    2:
        IF fbMotionDriveStateMachine.WatchDogTimeOut THEN
            nTestStep := nTestStep + 1;
        END_IF
    3:
        AssertEquals_INT(	Expected:=expectedMoveState,
                            Actual:=fbMotionDriveStateMachine.State,
                            Message:='Drive Machine state must be ERROR #1');
        AssertTrue(Condition := fbMotionDriveStateMachine.Error, Message := 'Motion Drive state machine must be in error state #2');
        nTestStep := nTestStep + 1;
        TEST_FINISHED();
END_CASE

fbMotionDriveStateMachine();
fbTestTimer();

IF fbTestTimer.Q THEN
    AssertTrue(Condition := FALSE, Message := CONCAT('Timed out at step: ', TO_STRING(nTestStep)));
    TEST_FINISHED();
END_IF
END_METHOD

METHOD PRIVATE GIvenStartedStatedAndErrorThenGotoErrorState_Test6
VAR_INST
    fbMotionDriveStateMachine : FB_MotionDriveStateMachine(
		stMotionCommand := THIS^.stMotionCommand[6],
		iMotionAxis:=THIS^.fbMotionAxisNC[6], 
		iMoveRequest:=THIS^.fbMoveRequest[6],
		iMotionLogger := THIS^.fbMotionLogger[6]
	);
    expectedMoveState : E_MoveState := E_MoveState.ERROR;

    nTestStep : INT;
END_VAR
TEST(__POUNAME());
CASE nTestStep OF
    0:
        fbMotionDriveStateMachine.State := E_MoveState.STARTED;
        fbMotionDriveStateMachine.StateMachine(Error:=TRUE);
        nTestStep := nTestStep + 1;
    1:
        AssertEquals_INT(	Expected:=expectedMoveState,
                            Actual:=fbMotionDriveStateMachine.State,
                            Message:='Drive Machine must be ERROR state #1');
        TEST_FINISHED();
END_CASE

fbMotionDriveStateMachine();
END_METHOD

END_FUNCTION_BLOCK

// ---- Test/TestDouble/FB_MotionAxisNC_TestDouble.TcPOU
FUNCTION_BLOCK FB_MotionAxisNC_TestDouble IMPLEMENTS I_MotionAxis
VAR

    iHome : I_Home;
    iHalt : I_Halt;
    iPower : I_Power;
    iReset : I_Reset;
    iMoveAbsolute : I_MoveAbsolute;
    iReadParameter : I_ReadParameter;
    iWriteParameter  : I_WriteParameter;
    iParamSaveRestore: I_ParamsSaveRestore;
    iEncoderScaling : I_EncoderScaling;
    iAxisStatus : I_AxisStatus;
    iBacklashCompensation : I_BacklashCompensation;

    bError: BOOL;
    nErrorID: UDINT;
    sMessage : T_MAXSTRING;
    stMotionAxisStatus : ST_AxisStatus;
END_VAR

METHOD AxisEnabled : BOOL
END_METHOD

(*
    Handle positive/negative backlash compensation
    User needs to set the direction of backlash from the sign of the compensation value
    Backlash compensation is disabled during referencing (homing).
    When direction is positive/negative, further movement in the negative/positive direction not compensated
    further movement in the negative/positive direction will be compensated
*)
METHOD BacklashCompensation
VAR_INPUT
    Enable	: BOOL := FALSE;
    RampVelo	: LREAL;
END_VAR
END_METHOD

METHOD ClearHaltStatus
END_METHOD

{warning 'Add method implementation '}
METHOD ClearHomeStatus
END_METHOD

{warning 'Add method implementation '}
METHOD ClearMoveAbsoluteStatus
END_METHOD

METHOD ClearResetStatus
END_METHOD

METHOD DisablePower
END_METHOD

METHOD DriveCommands
VAR_INPUT
    HomeCmd	: BOOL;
    NewMoveReq	: BOOL;
    EnableMode	: E_StageEnableMode;
END_VAR
END_METHOD

METHOD Halt
VAR_INPUT
    Deceleration	: LREAL := 0;
    Jerk	: LREAL := 0;
    BufferMode	: MC_BufferMode := MC_BufferMode.MC_Aborting;
END_VAR
END_METHOD

METHOD Home
VAR_INPUT
    Position        : LREAL         := DEFAULT_HOME_POSITION;
    BufferMode      : MC_BufferMode;
 	HomeMode: INT :=E_EpicsHomeCmd.NONE;
END_VAR
END_METHOD

{warning 'Add method implementation '}
METHOD HomeAbortRecovery
END_METHOD

METHOD MoveAbsolute
VAR_INPUT
    Position	: LREAL;
    Velocity	: LREAL;
    Acceleration	: LREAL := 0;
    Deceleration	: LREAL := 0;
    Jerk	: LREAL := 0;
    BufferMode	: MC_BufferMode := MC_BufferMode.MC_Aborting;
END_VAR
END_METHOD

METHOD Power
VAR_INPUT
    Enable	: BOOL;
    Enable_Positive	: BOOL;
    Enable_Negative	: BOOL;
    Override	: LREAL;
    BufferMode	: MC_BufferMode;
END_VAR
END_METHOD

METHOD ReadAxisParams
VAR_INPUT
    Enable	: BOOL;
    RefreshDelay	: TIME;
END_VAR
END_METHOD

METHOD Reset
END_METHOD

METHOD SaveAxisParams
VAR_INPUT
    Enable	: BOOL;
END_VAR
END_METHOD

PROPERTY Status : REFERENCE TO ST_AxisStatus
GET
Status REF= stMotionAxisStatus;
END_GET
END_PROPERTY

END_FUNCTION_BLOCK

// ---- Test/TestDouble/FB_MotionAxisDS402_TestDouble.TcPOU
FUNCTION_BLOCK FB_MotionAxisDS402_TestDouble IMPLEMENTS I_MotionAxisDS402
VAR
    bError: BOOL;
    nErrorID: UDINT;
    sMessage : T_MAXSTRING;
    stMotionAxisStatus : ST_AxisStatus;
    bConfigDone : BOOL;
END_VAR

METHOD AxisEnabled : BOOL
END_METHOD

(*
    Handle positive/negative backlash compensation
    User needs to set the direction of backlash from the sign of the compensation value
    Backlash compensation is disabled during referencing (homing).
    When direction is positive/negative, further movement in the negative/positive direction not compensated
    further movement in the negative/positive direction will be compensated
*)
METHOD BacklashCompensation
VAR_INPUT
    Enable	: BOOL := FALSE;
    RampVelo	: LREAL;
END_VAR
END_METHOD

METHOD ClearHaltStatus
END_METHOD

{warning 'Add method implementation '}
METHOD ClearHomeStatus
END_METHOD

{warning 'Add method implementation '}
METHOD ClearMoveAbsoluteStatus
END_METHOD

METHOD ClearResetStatus
END_METHOD

PROPERTY ConfigDone : BOOL
GET
ConfigDone := bConfigDone;
END_GET
SET
bConfigDone := ConfigDone;
END_SET
END_PROPERTY

METHOD DisablePower
END_METHOD

METHOD DriveCommands
VAR_INPUT
    HomeCmd	: BOOL;
    NewMoveReq	: BOOL;
    EnableMode	: E_StageEnableMode;
END_VAR
END_METHOD

METHOD Halt
VAR_INPUT
    Deceleration	: LREAL := 0;
    Jerk	: LREAL := 0;
    BufferMode	: MC_BufferMode := MC_BufferMode.MC_Aborting;
END_VAR
END_METHOD

METHOD Home
VAR_INPUT
    Position        : LREAL         := DEFAULT_HOME_POSITION;
    BufferMode      : MC_BufferMode;
 	HomeMode: INT :=E_EpicsHomeCmd.NONE;
END_VAR
END_METHOD

METHOD ModeConfigDone : BOOL
VAR_INPUT
    Mode	: E_EpicsMotorCmd;
END_VAR
 ModeConfigDone :=  bConfigDone;
END_METHOD

METHOD ModeOfOperation : BOOL
VAR_INPUT
    RecentModeOfOperation	: E_DS402OpMode;
END_VAR
END_METHOD

METHOD MoveAbsolute
VAR_INPUT
    Position	: LREAL;
    Velocity	: LREAL;
    Acceleration	: LREAL := 0;
    Deceleration	: LREAL := 0;
    Jerk	: LREAL := 0;
    BufferMode	: MC_BufferMode := MC_BufferMode.MC_Aborting;
END_VAR
END_METHOD

METHOD Power
VAR_INPUT
    Enable	: BOOL;
    Enable_Positive	: BOOL;
    Enable_Negative	: BOOL;
    Override	: LREAL;
    BufferMode	: MC_BufferMode;
END_VAR
END_METHOD

METHOD ReadAxisParams
VAR_INPUT
    Enable	: BOOL;
    RefreshDelay	: TIME;
END_VAR
END_METHOD

METHOD Reset
END_METHOD

METHOD SaveAxisParams
VAR_INPUT
    Enable	: BOOL;
END_VAR
END_METHOD

PROPERTY Status : REFERENCE TO ST_AxisStatus
GET
Status REF= stMotionAxisStatus;
END_GET
END_PROPERTY

END_FUNCTION_BLOCK

// ---- Test/TestDouble/FB_MoveRequest_TestDouble.TcPOU
FUNCTION_BLOCK FB_MoveRequest_TestDouble IMPLEMENTS I_MoveRequest
VAR
    eEnableMode: E_StageEnableMode:=E_StageEnableMode.DURING_MOTION;
    bMoveCmd	: BOOL;
    bHomeCmd: BOOL;
    eHomeMode	: E_EpicsHomeCmd;
    bEnableDone : BOOL;
    bMoveOk: BOOL;
    bExecute : BOOL;
    stMotionRequestStatus : ST_MoveRequestStatus;
END_VAR

METHOD ClearMoveRequest
END_METHOD

METHOD ClearMoveRequestErrors
END_METHOD

PROPERTY EnableMode : ENUM_StageEnableMode
GET
END_GET
SET
END_SET
END_PROPERTY

PROPERTY INTERNAL EpicsMotorCommand : INT
GET
EpicsMotorCommand := stMotionRequestStatus.nCommand;
END_GET
SET
stMotionRequestStatus.nCommand := EpicsMotorCommand;
END_SET
END_PROPERTY

METHOD HaltMoveRequest : BOOL
VAR_INPUT
    Busy	: BOOL;
END_VAR
END_METHOD

METHOD InitMoveRequest
END_METHOD

METHOD IsValidHomeCmd : BOOL
VAR_INPUT
    CmdData : INT;
END_VAR
END_METHOD

METHOD MoveRequest
VAR_INPUT
    (* From Axis through the drive*)
    EnableDone	: BOOL;
    (* From Interlock through the drive*)
    MoveOk	: BOOL;
END_VAR
END_METHOD

METHOD MoveRequestCompleted
VAR_INPUT
    MoveDone	: BOOL;
    HomeDone	: BOOL;
END_VAR
END_METHOD

METHOD MoveRequestDone
VAR_INPUT
    Done	: BOOL;
END_VAR
END_METHOD

METHOD MoveRequestError
VAR_INPUT
    Error	: BOOL;
    ErrorId	: UDINT;
    ErrorMessage	: T_MAXSTRING;
END_VAR
END_METHOD

METHOD MoveResetDone
END_METHOD

METHOD ResetMoveEnable : BOOL
END_METHOD

METHOD ResetMoveRequest
END_METHOD

METHOD RestoreSettings
VAR_INPUT
    RestoreDone : BOOL;
    SavedPosition : LREAL;
END_VAR
END_METHOD

PROPERTY Status : REFERENCE TO ST_MoveRequestStatus
GET
Status REF= stMotionRequestStatus;
END_GET
END_PROPERTY

{warning 'Add method implementation '}
METHOD StopMoveRequest
END_METHOD

END_FUNCTION_BLOCK

// ---- Test/Orchetration/FB_MotionDrive_Test.TcPOU
FUNCTION_BLOCK FB_MotionDrive_Test EXTENDS FB_TestSuite
VAR
	stMotionCommand : ST_MotionCommand;
    stMotionStatus: ST_MotionStatus;
	stExMotionStatus : ST_ExtendedMotionStatus;
    fbAxis         : FB_MotionAxisNC_TestDouble;        
    fbInterlocks   : FB_MotionInterlocksLimSw_TestDouble;  
    fbLogger       : FB_MotionLogger_TestDouble;      
    fbMoveRequest  : FB_MoveRequest_TestDouble;        
    fbStateMachine : FB_StateMachine_TestDouble;      
    fbBrake        : FB_Brake_TestDouble;              
END_VAR

NoCrashTest();

METHOD PRIVATE NoCrashTest
VAR_INST
	fbMotionDrive : FB_MotionDrive(	
		stMotionCommand :=stMotionCommand,
		stMotionStatus:=stMotionStatus,
		stExMotionStatus :=stExMotionStatus,
		iInterlocks :=fbInterlocks,
		iLogger :=fbLogger,
		iAxis:=fbAxis,
		iMoveRequest :=fbMoveRequest,
		iStateMachine :=fbStateMachine,
		iBrake :=fbBrake
	);


END_VAR
(*This method is called cyclicly in the fbMotionDrive *)
TEST(__POUNAME());
fbMotionDrive();
TEST_FINISHED();
END_METHOD

END_FUNCTION_BLOCK

// ---- Test/TestDouble/FB_MotionInterlocksLimSw_TestDouble.TcPOU
FUNCTION_BLOCK FB_MotionInterlocksLimSw_TestDouble IMPLEMENTS I_MotionInterlocks
VAR
END_VAR

METHOD AxisStatus
VAR_INPUT
    HomeBusy	: BOOL;
    PositiveDirection	: BOOL;
    NegativeDirection	: BOOL;
END_VAR
END_METHOD

METHOD DriveCommands
VAR_INPUT
    MoveEnable: BOOL;
    NewMoveReq : BOOL;
END_VAR
END_METHOD

PROPERTY Error : BOOL
GET
END_GET
END_PROPERTY

PROPERTY ErrorID : UDINT
GET
END_GET
END_PROPERTY

PROPERTY InterlockEvent : BOOL
GET
END_GET
END_PROPERTY

PROPERTY LimHome : BOOL
GET
END_GET
END_PROPERTY

PROPERTY Message : T_MAXSTRING
GET
END_GET
END_PROPERTY

PROPERTY MoveBackwardEnabled : BOOL
GET
END_GET
END_PROPERTY

PROPERTY MoveForwardEnabled : BOOL
GET
END_GET
END_PROPERTY

PROPERTY MoveOk : BOOL
GET
END_GET
END_PROPERTY

PROPERTY PowerEnabled : BOOL
GET
END_GET
END_PROPERTY

METHOD Reset
END_METHOD

PROPERTY Warning : BOOL
GET
END_GET
END_PROPERTY

END_FUNCTION_BLOCK

// ---- Test/TestDouble/FB_StateMachine_TestDouble.TcPOU
FUNCTION_BLOCK FB_StateMachine_TestDouble IMPLEMENTS I_StateMachine
VAR
END_VAR

{warning 'Add property implementation'}
PROPERTY Idling : BOOL
GET
END_GET
END_PROPERTY

PROPERTY MoveState : E_MOVESTATE
GET
END_GET
END_PROPERTY

{warning 'Add method implementation '}
METHOD Reset
END_METHOD

METHOD StateMachine
VAR_INPUT
	Error : BOOL;
	InterlockEvent : BOOL;
END_VAR
END_METHOD

PROPERTY WatchDogStatus : BOOL
GET
END_GET
END_PROPERTY

PROPERTY WatchDogTimeOut : BOOL
GET
END_GET
END_PROPERTY

END_FUNCTION_BLOCK

// ---- POUs/FBs/Common/FB_MotionDrive.TcPOU
FUNCTION_BLOCK FB_MotionDrive IMPLEMENTS I_MotionDrive
VAR_INPUT
END_VAR
VAR_OUTPUT
END_VAR
VAR
   // EPICS Interface
    {attribute 'no_copy'}
    stMotionEpicsItf : REFERENCE TO ST_MotionEpicsItf;
    {attribute 'hide'}
    iMotionAxis: I_MotionAxis;
    {attribute 'hide'}
    iBrake 				: I_Brake;
    {attribute 'hide'}
    iMotionInterlocks	: I_MotionInterlocks;
    {attribute 'hide'}
    iMotionLogger 		: I_MotionLogger;
    {attribute 'hide'}
    eMoveMode : E_EpicsMotorCmd := E_EpicsMotorCmd.MOVE_ABSOLUTE;
    // Determines when we automatically enable the motor
    //{attribute 'hide'}
    eEnableMode: E_StageEnableMode:=E_StageEnableMode.DURING_MOTION;

    (* Shortcut Commands *)
    // Start a move to fPosition with fVelocity
    bMoveCmd: BOOL;
    // Start the homing routine
    {attribute 'pytmc' := '
        pv: PLC:bHomeCmd
        io: io
        field: DESC Start the homing routine
    '}
    bHomeCmd: BOOL;
    // Close or open loop operation ( DS402 Piezo axis )
    {attribute 'pytmc' := '
        pv: PLC:bServo
        io: io
        field: ZNAM FALSE
        field: ONAM TRUE
        field: DESC Used internally to reset errors
    '}
    bServo : BOOL;

    sName : STRING;
    {attribute 'hide'}
    eMoveState	: E_MoveState;
    {attribute 'hide'}
    bNewMoveReq : BOOL;
    {attribute 'hide'}
    bExecHome 	: BOOL;
    {attribute 'hide'}
    bExecMove 	: BOOL;
    {attribute 'hide'}
    rtMoveCmdShortcut	: R_TRIG;
    {attribute 'hide'}
    rtHomeCmdShortcut 	: R_TRIG;
    {attribute 'hide'}
    rtUserExec 			: R_TRIG;
    {attribute 'hide'}
    rtNewMoveReq 		: R_TRIG;
    {attribute 'hide'}
    rtTarget			: R_TRIG;
    {attribute 'hide'}
    rtHomed				: R_TRIG;
    {attribute 'hide'}
    rtValidExec 	: R_TRIG;
    {attribute 'hide'}
    rtReset 			: R_TRIG;
    {attribute 'hide'}
    ftStopExec 			: F_TRIG;
    {attribute 'hide'}
    ftError 			: F_TRIG;
    {attribute 'hide'}
    nCommandLocal: UINT;
    {attribute 'hide'}
    nCmdDataLocal: UINT;
    {attribute 'hide'}
    ftLocalStart : F_TRIG;
    {attribute 'hide'}
    bInitStart : BOOL;
    {attribute 'hide'}
    bLocalExec : BOOL;
    {attribute 'hide'}
    bEnableDone : BOOL;
    {attribute 'hide'}
    bPrepareDisable : BOOL;
    {attribute 'hide'}
    rtEnableMode : R_TRIG;
    {attribute 'hide'}
    rtStopExec : R_TRIG;
    {attribute 'hide'}
    rtInterlockEvent : R_TRIG;
    {attribute 'hide'}
    bCmdExecute : BOOL;
    {attribute 'hide'}
    bHaltAbort : BOOL;
    {attribute 'hide'}
    ftHaltAbort : F_TRIG;
    {attribute 'hide'}
    rtRestoreDone : R_TRIG;
    {attribute 'hide'}
    bHaltEvent : BOOL;
    // move state machine to error state in case a move command gets stuck after
    // the corresponding start signal was forwarded. the start signal should yeild a busy true response.
    // the move processing block may get stuck and return no errors. this is a contingency to make sure that reset would reinit all state machines.
    tonSyncTimer : TON;
    bLocalError : BOOL;
    bLocalMessage : T_MAXSTRING;
END_VAR

IF NOT __ISVALIDREF( THIS^.stMotionEpicsItf ) THEN
   RETURN;
END_IF
// Restore axis parameters
THIS^.RestoreSettings();

// catch high priority message
// an extended error message from FB_MotionLogger will display cyclic errors and warning
IF iMotionAxis.Error THEN
   stMotionEpicsItf.bError := iMotionAxis.Error;
   stMotionEpicsItf.nErrorId := iMotionAxis.ErrorID;
   stMotionEpicsItf.sErrorMessage := iMotionAxis.Message;
ELSIF iMotionInterlocks.Error THEN
   stMotionEpicsItf.bError := iMotionInterlocks.Error;
   stMotionEpicsItf.nErrorId := iMotionInterlocks.ErrorID;
   stMotionEpicsItf.sErrorMessage := iMotionInterlocks.Message;
ELSIF bLocalError THEN
   stMotionEpicsItf.bError := bLocalError;
   stMotionEpicsItf.sErrorMessage := bLocalMessage;
// Warnings have lowest priority
ELSIF iMotionInterlocks.Warning THEN
   stMotionEpicsItf.sErrorMessage := iMotionInterlocks.Message;
ELSE
       stMotionEpicsItf.bError := FALSE;
       stMotionEpicsItf.nErrorId := 0;
       stMotionEpicsItf.sErrorMessage := '';

END_IF

// Drive state machine
THIS^.StateMachine();
//
THIS^.PostHandling();
// update EPICS status
THIS^.UpdateParamAndStatus();

METHOD PUBLIC CallAfterInit
VAR_INPUT
    stMotionEpicsItf : REFERENCE TO ST_MotionEpicsItf;
    iBrake : I_Brake;
    iMotionInterlocks : I_MotionInterlocks;
    iMotionLogger : I_MotionLogger;
    iMotionAxis: I_MotionAxis;
END_VAR
THIS^.stMotionEpicsItf REF=stMotionEpicsItf;
THIS^.iMotionAxis := iMotionAxis;
THIS^.iMotionLogger:=iMotionLogger;
THIS^.iBrake:=iBrake;
THIS^.iMotionInterlocks:=iMotionInterlocks;
END_METHOD

METHOD ClearVars
VAR_INPUT
    Done : BOOL;
END_VAR
stMotionEpicsItf.bDone := Done;
stMotionEpicsItf.bBusy := FALSE;
// falling edge here when target is reached, move halted
stMotionEpicsItf.bExecute := FALSE;
THIS^.bLocalExec := FALSE;
// release the cmds
THIS^.bHomeCmd:=FALSE;
THIS^.bMoveCmd:=FALSE;
THIS^.binitStart := FALSE;
THIS^.bCmdExecute := FALSE;
THIS^.tonSyncTimer.IN:=FALSE;
END_METHOD

{warning 'Add property implementation'}
PROPERTY EnableMode : ENUM_StageEnableMode
GET
EnableMode := eEnableMode;
END_GET
SET
eEnableMode := EnableMode;
END_SET
END_PROPERTY

//FB_Init is always available implicitly and it is used primarily for initialization.
//The return value is not evaluated. For a specific influence, you can also declare the
//methods explicitly and provide additional code there with the standard initialization
//code. You can evaluate the return value.
METHOD FB_Init: BOOL
VAR_INPUT
    bInitRetains: BOOL; // TRUE: the retain variables are initialized (reset warm / reset cold)
    bInCopyCode: BOOL;  // TRUE: the instance will be copied to the copy code afterward (online change)
    stMotionEpicsItf : REFERENCE TO ST_MotionEpicsItf;
    iBrake : I_Brake;
    iMotionInterlocks : I_MotionInterlocks;
    iMotionLogger : I_MotionLogger;
    iMotionAxis: I_MotionAxis;
   // iLimSwStatus : I_LimSwStatus;
END_VAR
THIS^.stMotionEpicsItf REF=stMotionEpicsItf;
THIS^.iMotionAxis := iMotionAxis;
THIS^.iMotionLogger:=iMotionLogger;
THIS^.iBrake:=iBrake;
//THIS^.iLimSwStatus:=iLimSwStatus;
THIS^.iMotionInterlocks:=iMotionInterlocks;
END_METHOD

{attribute 'call_after_init'}
METHOD Instances
VAR_INPUT
END_VAR

VAR

END_VAR
// bMotionAxisNC  := __QUERYINTERFACE(iMotionAxisCommon, iMotionAxisNC) AND NOT __QUERYINTERFACE(iMotionAxisCommon,iMotionAxisCommonDS402);
// bMotionAxisNCDS402  := __QUERYINTERFACE(iMotionAxisCommon,iMotionAxisNCDS402) AND __QUERYINTERFACE(iMotionAxisCommon,iMotionAxisCommonDS402);
// bMotionAxisDS402  := __QUERYINTERFACE(iMotionAxisCommon, iMotionAxisDS402);
// bMotionInterlocks  := __QUERYINTERFACE(iMotionInterlocks,iMotionInterlocks) AND NOT __QUERYINTERFACE(iMotionInterlocks,iLimSw);
// bMotionInterlocksLimSw  := __QUERYINTERFACE(iMotionInterlocks,iMotionInterlocks) AND __QUERYINTERFACE(iMotionInterlocks,iLimSw);;
END_METHOD

{warning 'Add property implementation'}
PROPERTY Name : STRING
GET
Name := sName;
END_GET
SET
sName := Name;
END_SET
END_PROPERTY

{warning 'Add method implementation '}
METHOD PostHandling
// Move done, or aborted? prepare disable.
// we'll wait for axis to be in standstill and this state machine to be idling.
THIS^.bPrepareDisable S= (eEnableMode = E_StageEnableMode.DURING_MOTION ) AND THIS^.ftStopExec.Q;
//
// IF THIS^.stMotionEpicsItf.bReset THEN
//    // Relese motion cmds
//    THIS^.ClearVars(Done:=FALSE);
//  			THIS^.bLocalError := FALSE;
// 			THIS^.bLocalMessage := '';
//    // Forward general reset event
//    THIS^.iMotionAxis.Reset(Execute:= THIS^.stMotionEpicsItf.bReset);
//    THIS^.stMotionEpicsItf.bReset := FALSE;
// END_IF

// When reset is done axis is standstill
// safe to remove power
IF iMotionAxis.ResetDone THEN
    THIS^.stMotionEpicsItf.bEnable := FALSE;
END_IF

// Default is move absolute for state psotioner
IF THIS^.rtHomed.Q THEN
       stMotionEpicsItf.nCommand:=E_EpicsMotorCmd.MOVE_ABSOLUTE;
END_IF
// Halt is always a user stop but not an interlock event or a reset.
bHaltEvent S= ftStopExec.Q AND ((iMotionAxis.HomeBusy AND (nCommandLocal=10))
                            OR(iMotionAxis.MoveAbsoluteBusy AND (nCommandLocal=3)));
bHaltEvent R= THIS^.iMotionAxis.HaltDone OR THIS^.iMotionAxis.ResetDone;

THIS^.iMotionAxis.Halt(	Execute:=bHaltEvent,
                        Deceleration:=stMotionEpicsItf.fDeceleration);

//
THIS^.iMotionInterlocks.AxisStatus(
                            HomeBusy:=THIS^.iMotionAxis.HomeBusy,
                            PositiveDirection:=THIS^.iMotionAxis.PositiveMotionIsEnabled,
                            NegativeDirection:=THIS^.iMotionAxis.NegativeMotionIsEnabled );

// Forward drive commands to interlock blocks
THIS^.iMotionInterlocks.DriveCommands(Enable:=THIS^.stMotionEpicsItf.bEnable, NewMoveReq:=THIS^.bNewMoveReq, Reset:=THIS^.iMotionAxis.ResetDone);
// Forward Power block enable flags
THIS^.iMotionAxis.PowerEnables(Enable:=iMotionInterlocks.PowerEnabled,
                        Enable_Positive:=iMotionInterlocks.MoveForwardEnabled,
                        Enable_Negative:=iMotionInterlocks.MoveBackwardEnabled );

// Forward axis state to brake FB
THIS^.iBrake.AxisState := iMotionAxis.AxisState;

// Read Axis Parameter
THIS^.iMotionAxis.ReadAxisParams(Enable:=TRUE, RefreshDelay:=T#1S);

// Save and Restore
THIS^.iMotionAxis.SaveAxisParams(Enable:=TRUE);
END_METHOD

METHOD PreHandling
(*
  Check for the plc shortcut commands
  Used for testing or to circumvent motor record issues
  A request is process and qualified as a legitimate move after it clears interlocks checks
*)
rtMoveCmdShortcut(CLK:=THIS^.bMoveCmd);
rtHomeCmdShortcut(CLK:=THIS^.bHomeCmd);
// Execute on rising edge
IF rtMoveCmdShortcut.Q AND NOT stMotionEpicsItf.bExecute THEN
   stMotionEpicsItf.bExecute:=TRUE;
   stMotionEpicsItf.nCommand:=E_EpicsMotorCmd.MOVE_ABSOLUTE;
   // attempting to move an axis without homing first?
   IF iMotionAxis.HomeMode <> E_EpicsHomeCmd.NONE AND NOT iMotionAxis.HomeDone THEN
       stMotionEpicsItf.sErrorMessage:='Axis homing mode set, but homing routine pending';
   END_IF
ELSIF rtHomeCmdShortcut.Q AND NOT stMotionEpicsItf.bExecute THEN
       stMotionEpicsItf.nCommand:=E_EpicsMotorCmd.HOME;
       // Automatically fill the correct nCmdData for homing
       stMotionEpicsItf.nCmdData:=iMotionAxis.HomeMode;
       IF ( stMotionEpicsItf.nCmdData = E_EpicsHomeCmd.ABSOLUTE_SET )  OR ( stMotionEpicsItf.nCmdData = E_EpicsHomeCmd.NONE) THEN
       stMotionEpicsItf.bExecute:= FALSE;
       THIS^.bHomeCmd := FALSE;
    ELSE
        stMotionEpicsItf.bExecute:= TRUE;
    END_IF
END_IF

rtUserExec(CLK:=stMotionEpicsItf.bExecute);
bNewMoveReq S= rtUserExec.Q AND NOT iMotionAxis.Busy AND iMotionInterlocks.MoveOk;
// An axis or interlocks error will immediately invalidate this this request.
bNewMoveReq R= NOT stMotionEpicsItf.bExecute OR stMotionEpicsItf.bError;
bPrepareDisable R= bNewMoveReq;
//
rtNewMoveReq(CLK:=bNewMoveReq);
rtEnableMode(CLK:=(eEnableMode = E_StageEnableMode.DURING_MOTION));
// Handle auto-enable timing
CASE eEnableMode OF
   E_StageEnableMode.ALWAYS:
       stMotionEpicsItf.bEnable:=TRUE;
   E_StageEnableMode.DURING_MOTION:
       IF rtEnableMode.Q THEN
           stMotionEpicsItf.bEnable := FALSE;
       END_IF
       // Power interlock only enabled with a new move request
       IF rtNewMoveReq.Q THEN
           stMotionEpicsItf.bEnable S= bNewMoveReq (*iMotionInterlocks.SafetyReady*);
       END_IF
END_CASE
//
// Get a definitive bEnabled reading
THIS^.bEnableDone := THIS^.iMotionAxis.AxisEnabled(HomeCmd:=THIS^.bHomeCmd, NewMoveReq:=THIS^.bNewMoveReq);

// This is the output interlock check used to allow the requested move
bLocalExec:= stMotionEpicsItf.bExecute AND iMotionInterlocks.PowerEnabled AND THIS^.bEnableDone (*AND iMotionInterlocks.SafetyReady*);

bExecHome:=THIS^.bLocalExec AND stMotionEpicsItf.nCommand = 10;
bExecMove:=THIS^.bLocalExec AND NOT bExecHome;
//
// Transfer nCommand and nCmdData to local copies at rising edge of bExecute
// (avoid issues if nCommand or nCmdData are changed during a command)
rtValidExec(CLK:=(THIS^.bExecMove OR THIS^.bExecHome));
IF rtValidExec.Q THEN
 // used for jog, modulo, GearIn which are not implemented here
 nCmdDataLocal:=INT_TO_UINT(stMotionEpicsItf.nCmdData);
 nCommandLocal:=INT_TO_UINT(stMotionEpicsItf.nCommand);
END_IF
END_METHOD

METHOD RestoreSettings
VAR_INPUT
END_VAR
// no needed in production since the actualposition is already set on the axis
// and epics status will get that last position
// use this to restore anything thats not an axisref paramter.
rtRestoreDone(CLK:= THIS^.iMotionAxis.RestoreDone);
IF rtRestoreDone.Q THEN
    THIS^.stMotionEpicsItf.fPosition := THIS^.iMotionAxis.SavedPosition;
END_IF
END_METHOD

{warning 'Add method implementation '}
METHOD StateMachine
ftError(CLK:=stMotionEpicsItf.bError);
rtTarget(CLK:=(iMotionAxis.MoveAbsoluteDone AND bExecMove));
rtHomed(CLK:=iMotionAxis.HomeDone (* AND bExecHome*));
ftStopExec(CLK:=stMotionEpicsItf.bExecute);
//
rtInterlockEvent(CLK:=iMotionInterlocks.InterlockEvent);
rtReset(CLK:=stMotionEpicsItf.bReset);
IF rtReset.Q OR rtInterlockEvent.Q THEN
    IF THIS^.stMotionEpicsItf.bReset THEN
        // Relese motion cmds
        THIS^.ClearVars(Done:=FALSE);
        THIS^.bLocalError := FALSE;
        THIS^.bLocalMessage := '';
        // Forward general reset event
        THIS^.iMotionAxis.Reset(Execute:= THIS^.stMotionEpicsItf.bReset);
        THIS^.stMotionEpicsItf.bReset := FALSE;
    END_IF
    stMotionEpicsItf.bExecute := FALSE;
END_IF

// Drive state Machine here
CASE eMoveState OF
   E_MoveState.IDLING:
        THIS^.PreHandling();
        // Delay the disable until axis reach standstill
        // and this state machine is idling
        IF THIS^.bPrepareDisable AND THIS^.iMotionAxis.StandStill THEN
            THIS^.bPrepareDisable := FALSE;
            THIS^.stMotionEpicsItf.bEnable := FALSE;
        ELSIF bExecMove OR bExecHome THEN
               eMoveState := E_MoveState.INIT;
        ELSIF stMotionEpicsItf.bError THEN
               eMoveState := E_MoveState.ERROR;
        END_IF

   E_MoveState.INIT:
       // When we start, set the busy/done appropriately
       stMotionEpicsItf.bBusy := TRUE;
       stMotionEpicsItf.bDone := FALSE;
       // reset error flag
       stMotionEpicsItf.sErrorMessage := '';
       CASE stMotionEpicsItf.nCommand OF
           E_EpicsMotorCmd.MOVE_ABSOLUTE:
               eMoveMode := E_EpicsMotorCmd.MOVE_ABSOLUTE;
               bCmdExecute := bExecMove AND (nCommandLocal=3);
           E_EpicsMotorCmd.HOME:
               eMoveMode := E_EpicsMotorCmd.HOME;
               bCmdExecute := nCommandLocal=10 AND bExecHome;
       END_CASE

       IF bExecMove THEN
            THIS^.iMotionAxis.MoveAbsolute(	Execute:=FALSE,
                       Position:=THIS^.stMotionEpicsItf.fPosition,
                       Velocity := THIS^.stMotionEpicsItf.fVelocity,
                       Acceleration := THIS^.stMotionEpicsItf.fAcceleration,
                       Deceleration := THIS^.stMotionEpicsItf.fDeceleration
                );
            // Activate backlash compensation
            THIS^.iMotionAxis.BacklashCompensationActive(Active:=TRUE, RampVelocity:=THIS^.stMotionEpicsItf.fVelocity/10.0);
       ELSIF bExecHome THEN
            // Deactivate backlash compensation
            THIS^.iMotionAxis.BacklashCompensationActive(Active:=FALSE, RampVelocity:=0.0);
       END_IF

       iMotionAxis.StartMove( eMoveMode, bCmdExecute );
       // configure and start move.
       tonSyncTimer.IN:=TRUE;
        eMoveState := E_MoveState.STARTED;
   E_MoveState.STARTED:
       IF stMotionEpicsItf.bError THEN
           eMoveState := E_MoveState.ERROR;
        // Move Started? use a timer to force quit this state if no response from axis
       ELSIF tonSyncTimer.Q THEN
           bLocalError := TRUE;
           bLocalMessage := 'No Response from Axis';
           eMoveState := E_MoveState.ERROR;
       ELSIF iMotionAxis.Busy THEN
           eMoveState := E_MoveState.IN_PROGRESS;
       END_IF

   E_MoveState.IN_PROGRESS :

       IF 	stMotionEpicsItf.bError THEN
           eMoveState := E_MoveState.ERROR;

       // Move interupted
       ELSIF ftStopExec.Q OR iMotionAxis.Aborted THEN
           eMoveState := E_MoveState.INTERRUPTED;

       ELSIF  rtTarget.Q OR rtHomed.Q  THEN
           eMoveState := E_MoveState.REACHED;
       END_IF

   E_MoveState.INTERRUPTED:

       IF THIS^.iMotionInterlocks.InterlockEvent THEN
           eMoveState := E_MoveState.REACHED;
       END_IF
       // Wait here for halt or reset done or clearing limit state to be restored
       IF iMotionAxis.AbortDone THEN
           THIS^.ClearVars(Done:=TRUE);
           eMoveState := E_MoveState.IDLING;;
       END_IF

   E_MoveState.REACHED:
       THIS^.ClearVars(Done:=TRUE);
       eMoveState := E_MoveState.IDLING;

   E_MoveState.ERROR:
       THIS^.ClearVars(Done:=FALSE);
       THIS^.stMotionEpicsItf.bEnable := FALSE;

       IF ftError.Q THEN
           eMoveState := E_MoveState.IDLING;
       END_IF

END_CASE
// the wait time is about 5 plc task cycle
 tonSyncTimer(PT:=T#60S);
END_METHOD

METHOD UpdateParamAndStatus

//////////////////////////////////////////////////////////////////
// Transfer NC parameter status to EPICS
//////////////////////////////////////////////////////////////////
stMotionEpicsItf.stAxisStatus.bEnable:=iMotionInterlocks.PowerEnabled;
stMotionEpicsItf.stAxisStatus.bEnabled:=iMotionAxis.PowerIsEnabled;
stMotionEpicsItf.stAxisStatus.bExecute:=THIS^.bLocalExec;
stMotionEpicsItf.stAxisStatus.bHomeSensor:=iMotionInterlocks.LimHome;

stMotionEpicsItf.stAxisStatus.bLimitBwd:= iMotionInterlocks.MoveBackwardEnabled;
stMotionEpicsItf.stAxisStatus.bLimitFwd:= iMotionInterlocks.MoveForwardEnabled;
stMotionEpicsItf.stAxisStatus.fActDiff:=iMotionAxis.MeasuredPositionDiff;
stMotionEpicsItf.stAxisStatus.fActPosition:=iMotionAxis.MeasuredPosition;
stMotionEpicsItf.stAxisStatus.fActVelocity:=iMotionAxis.MeasuredVelocity;
stMotionEpicsItf.stAxisStatus.fOverride:=iMotionAxis.PowerOverride;
stMotionEpicsItf.stAxisStatus.bBusy:=iMotionAxis.Busy;
stMotionEpicsItf.stAxisStatus.bHomed:=iMotionAxis.HomeDone;
//stMotionEpicsInterface.stAxisStatus.bJogBwd:=bJogBwd;
//stMotionEpicsInterface.stAxisStatus.bJogFwd:=bJogFwd;
stMotionEpicsItf.stAxisStatus.bReset:=stMotionEpicsItf.bReset;
stMotionEpicsItf.stAxisStatus.bError:=stMotionEpicsItf.bError;
stMotionEpicsItf.stAxisStatus.fAcceleration:=stMotionEpicsItf.fAcceleration;
stMotionEpicsItf.stAxisStatus.fDeceleration:=stMotionEpicsItf.fDeceleration;
stMotionEpicsItf.stAxisStatus.fPosition:=stMotionEpicsItf.fPosition;
stMotionEpicsItf.stAxisStatus.fVelocity:=stMotionEpicsItf.fVelocity;
stMotionEpicsItf.stAxisStatus.nCmdData:=INT_TO_UINT(stMotionEpicsItf.nCmdData);  //Or nCmdDataLocal
stMotionEpicsItf.stAxisStatus.nCommand:=INT_TO_UINT(stMotionEpicsItf.nCommand);  //Or nCommandLocal
stMotionEpicsItf.stAxisStatus.nErrorId:=stMotionEpicsItf.nErrorId;
END_METHOD

END_FUNCTION_BLOCK

// ---- Test/NC/FB_NcMotionBlocks_Test.TcPOU
FUNCTION_BLOCK FB_NcMotionBlocks_Test EXTENDS FB_TestSuite
VAR
    fbAxisRef : ARRAY [1..16] OF AXIS_REF;
    fbLimSwStatus : ARRAY [1..16] OF FB_LimSwStatus_TestDouble;
    fbMotionLogger : ARRAY [1..16] OF FB_MotionLogger_TestDouble;
    fbPower : ARRAY [1..16] OF FB_PowerNC[	(AxisRef := fbAxisRef[1], iMotionLogger:= fbMotionLogger[1]),
                                            (AxisRef := fbAxisRef[2], iMotionLogger:= fbMotionLogger[2]),
                                            (AxisRef := fbAxisRef[3], iMotionLogger:= fbMotionLogger[3]),
                                            (AxisRef := fbAxisRef[4], iMotionLogger:= fbMotionLogger[4]),
                                            (AxisRef := fbAxisRef[5], iMotionLogger:= fbMotionLogger[5]),
                                            (AxisRef := fbAxisRef[6], iMotionLogger:= fbMotionLogger[6]),
                                            (AxisRef := fbAxisRef[7], iMotionLogger:= fbMotionLogger[7]),
                                            (AxisRef := fbAxisRef[8], iMotionLogger:= fbMotionLogger[8]),
											(AxisRef := fbAxisRef[9], iMotionLogger:= fbMotionLogger[9]),
                                            (AxisRef := fbAxisRef[10], iMotionLogger:= fbMotionLogger[10]),
                                            (AxisRef := fbAxisRef[11], iMotionLogger:= fbMotionLogger[11]),
                                            (AxisRef := fbAxisRef[12], iMotionLogger:= fbMotionLogger[12]),
                                            (AxisRef := fbAxisRef[13], iMotionLogger:= fbMotionLogger[13]),
                                            (AxisRef := fbAxisRef[14], iMotionLogger:= fbMotionLogger[14]),
                                            (AxisRef := fbAxisRef[15], iMotionLogger:= fbMotionLogger[15]),
                                            (AxisRef := fbAxisRef[16], iMotionLogger:= fbMotionLogger[16])
                                            ];
END_VAR

GivenHomeCmdAbsoluteSetModeThenSetHomeDoneAndPositionToUserDefineOffset_Test1();
GivenHomeCmdBacklashCompensationInactiveThenMoveStartandCompletesWithBacklashCompensationDisabled_Test2();
GivenHomeCmdHomeViaHighModeAndHomeSwPulseThenMoveToUserDefineOffset_Test3();
GivenHomeCmdHomeViaHighModeForwardSwPulseBeforeHomeSwPulseThenMoveToUserDefineOffset_Test4();
GivenHomeCmdHomeViaLowModeAndHomeSwPulseThenMoveToUserDefineOffset_Test5();
GivenHomeCmdHomeViaLowModeBackwardSwPulseBeforeHomeSwPulseThenMoveToUserDefineOffset_Test6();
GivenHomeCmdLowLimitModeAndABackwardSwPulseThenHomeDoneAndPositionSetToUserDefineOffset_Test7();
GivenHomeCmdNoneModeThenSetHomeFlag_Test8();
GivenHomeCmdSetToHighLimitAndHighLimitPulseThenSetHomeDoneAndPositionToUserDefineOffset_Test9();
GivenMoveCmdNegativeBacklashCompensationActiveThenReverseMoveIsCompensated_Test10();
GivenMoveCmdPositiveBacklashCompensationActiveThenReverseMoveIsCompensated_Test11();
GivenDirectionalPowerEnabledAndBackwardAbsoluteMoveIfNegativeLimitHitThenAbortMove_Test12();
GivenDirectionalPowerEnabledAndForwardAbsoluteMoveIfPositiveLimitHitThenAbortMove_Test13();
GivenPowerIsEnabledAndCompletedAbsoluteMoveThenMoveAbsoluteDoneStatusRetained_Test14();
GivenPowerIsEnabledAndAbsoluteMoveStartedIfHaltSignalThenMoveIsAbortedAndHaltDoneIsRetained_Test15();
GivenPowerIsEnabledAbsoluteMoveIfResetThenMoveIsAbortedAndResetDoneIsRetained_Test16();

//

METHOD PRIVATE GivenDirectionalPowerEnabledAndBackwardAbsoluteMoveIfNegativeLimitHitThenAbortMove_Test12
VAR_INST
    // Subject under tests
    fbMoveAbsolute : FB_MoveAbsoluteNC(AxisRef := fbAxisRef[12],  iMotionLogger:= fbMotionLogger[12]);
    fbTestTimer : TON := (PT := T#3S, IN := TRUE);
    nTestStateStep : INT;
    fbLimtHitTimer : TON := (PT := T#1S, IN := FALSE);
    fExpectedPosition: LREAL := 50.0;
END_VAR
TEST(__POUNAME());

// Cyclically call these every scan for correct PLC logic
fbPower[12].Power(
    Enable := TRUE,
    Enable_Positive := fbLimSwStatus[12].LimitForwardEnable,
    Enable_Negative := fbLimSwStatus[12].LimitBackwardEnable,
    Override := 100
);

// Stepwise state machine logic
CASE nTestStateStep OF
    0 : // Wait for power on before initiating move
        IF fbPower[12].PowerIsEnabled THEN
            nTestStateStep := 1;
        END_IF

    1 : // Issue negative move and start timer
        fbMoveAbsolute.MoveAbsolute(
            Position := -150.0,
            Velocity := 100,
            Acceleration := 200,
            Deceleration := 200
        );
        fbLimtHitTimer.IN := TRUE;
        nTestStateStep := 2;

    2 : // After timer, simulate limit hit
        IF fbLimtHitTimer.Q THEN
            fbLimSwStatus[12].LimitBackwardEnable := FALSE; // Simulate the axis hitting the negative limit
            nTestStateStep := 3;
        END_IF

    3 : // Wait until move is aborted by limit hit
        IF fbMoveAbsolute.Aborted THEN
            nTestStateStep := 4;
        END_IF

    4 : // Assertions below once test finished
END_CASE

// Cyclic calls required for correct behavior
fbLimtHitTimer();
fbTestTimer();
fbAxisRef[12].ReadStatus();
fbMoveAbsolute();

// Final assertion and test finish
IF nTestStateStep = 4 THEN
    AssertTrue(
        Condition := fbAxisRef[12].Status.HasBeenStopped,
        Message := 'Expected HasBeenStopped after move aborted by limit'
    );
    TEST_FINISHED();

ELSIF fbTestTimer.Q THEN
    AssertTrue(
        Condition := FALSE,
        Message := CONCAT('Timed out at step: ', TO_STRING(nTestStateStep))
    );
    TEST_FINISHED();
END_IF
END_METHOD

METHOD PRIVATE GivenDirectionalPowerEnabledAndForwardAbsoluteMoveIfPositiveLimitHitThenAbortMove_Test13
VAR_INST

    // Subject under tests
    fbMoveAbsolute : FB_MoveAbsoluteNC(AxisRef := fbAxisRef[13], iMotionLogger:= fbMotionLogger[13]);
    fbTestTimer : TON := (PT := T#3S, IN := TRUE);
    nTestStateStep : INT;
    fbLimtHitTimer : TON := (PT := T#1S, IN := FALSE);
    fExpectedPosition: LREAL := 50.0;
END_VAR
TEST(__POUNAME());

// Cyclically call these every scan for correct PLC logic
fbPower[13].Power(
    Enable := TRUE,
    Enable_Positive := fbLimSwStatus[13].LimitForwardEnable,
    Enable_Negative := fbLimSwStatus[13].LimitBackwardEnable,
    Override := 100
);

// Stepwise state machine logic
CASE nTestStateStep OF
    0 : // Wait for power on before initiating move
        IF fbPower[13].PowerIsEnabled THEN
            nTestStateStep := 1;
        END_IF

    1 : // Issue negative move and start timer
        fbMoveAbsolute.MoveAbsolute(
            Position := 150.0,
            Velocity := 100,
            Acceleration := 200,
            Deceleration := 200
        );
        fbLimtHitTimer.IN := TRUE;
        nTestStateStep := 2;

    2 : // After timer, simulate limit hit
        IF fbLimtHitTimer.Q THEN
            fbLimSwStatus[13].LimitForwardEnable := FALSE; // Simulate the axis hitting the negative limit
            nTestStateStep := 3;
        END_IF

    3 : // Wait until move is aborted by limit hit
        IF fbMoveAbsolute.Aborted THEN
            nTestStateStep := 4;
        END_IF
END_CASE

// Cyclic calls required for correct behavior
fbLimtHitTimer();
fbTestTimer();
fbAxisRef[13].ReadStatus();
fbMoveAbsolute();

// Final assertion and test finish
IF nTestStateStep = 4 THEN
    AssertTrue(
        Condition := fbAxisRef[13].Status.HasBeenStopped,
        Message := 'Expected HasBeenStopped after move aborted by limit'
    );
    TEST_FINISHED();

ELSIF fbTestTimer.Q THEN
    AssertTrue(
        Condition := FALSE,
        Message := CONCAT('Timed out at step: ', TO_STRING(nTestStateStep))
    );
    TEST_FINISHED();
END_IF
END_METHOD

METHOD PRIVATE GivenHomeCmdAbsoluteSetModeThenSetHomeDoneAndPositionToUserDefineOffset_Test1
VAR_INST
    fbHome : FB_HomeNC(
		AxisRef:=fbAxisRef[1],
		iLimSwStatus:=fbLimSwStatus[1],
		iMotionLogger:=fbMotionLogger[1]
	):=(Mode:=E_EpicsHomeCmd.ABSOLUTE_SET);
    fbTestTimer : TON := (IN := TRUE, PT := T#8S);
    nTestStep : INT := 0;
    fExpectedPosition : LREAL := 20.0;
    fActPosition : LREAL := 0.0;
    bCalibrated : BOOL := FALSE;
END_VAR
TEST(__POUNAME());
// FBs that must be invoked cyclically
fbLimSwStatus[1]();
fbMotionLogger[1]();
fbAxisRef[1].ReadStatus();
fbPower[1].Power(
    Enable := TRUE,
    Enable_Positive := fbLimSwStatus[1].LimitForwardEnable,
    Enable_Negative := fbLimSwStatus[1].LimitBackwardEnable,
    Override := 100.0
);
fbHome();
fbTestTimer(IN := TRUE);

// --- State Machine ---
CASE nTestStep OF
    0: // Enable power, then issue home command
        IF fbPower[1].PowerIsEnabled THEN
            fbHome.Home(Position := fExpectedPosition, BufferMode := MC_BufferMode.MC_Aborting);
            nTestStep := 1;
        END_IF

    1: // Wait for homing to complete
        IF fbHome.Done THEN
            nTestStep := 2;
        END_IF
END_CASE

// --- Test Completion: Assertion & Finish ---
IF nTestStep = 2 THEN
    bCalibrated := fbHome.Done;

    // Assert the axis is marked homed (calibrated)
    AssertEquals_BOOL(
        Expected := TRUE,
        Actual := fbAxisRef[1].Status.Homed,
        Message := 'Axis not calibrated #1'
    );

    // Assert the position matches expected
    AssertEquals_LREAL(
        Delta := 0.001,
        Expected := fExpectedPosition,
        Actual := fbAxisRef[1].NcToPlc.ActPos,
        Message := 'Position is not the expected #2'
    );
    TEST_FINISHED();

ELSIF fbTestTimer.Q THEN
    AssertTrue(
        Condition := FALSE,
        Message := CONCAT('Timed out at step: ', TO_STRING(nTestStep))
    );
    TEST_FINISHED();
END_IF
END_METHOD

METHOD PRIVATE GivenHomeCmdBacklashCompensationInactiveThenMoveStartandCompletesWithBacklashCompensationDisabled_Test2
VAR_INST

    // Subjects under tests
    fbBacklashCompensation : FB_BacklashCompensationNC(
		AxisRef := fbAxisRef[2], 
		iMotionLogger:= fbMotionLogger[2]
	);

    fbHome : FB_HomeNC(
		AxisRef:=fbAxisRef[2],
		iLimSwStatus:=fbLimSwStatus[2],
		iMotionLogger:=fbMotionLogger[2]
	):=(Mode:=E_EpicsHomeCmd.HIGH_LIMIT);

    fbTestTimer : TON := (PT := T#5S, IN := TRUE);
    nTestStep : INT;
    fbCamSwitchPulserSearch: TON := (IN:=TRUE, PT:=T#100MS);
    fbCamSwitchPulserSync: TON := (PT:=T#500MS);
    bHomingOverride: BOOL := TRUE;

END_VAR
TEST(__POUNAME());

// Directional enables must always be TRUE during homing via override.
// 'bHomingOverride' should be TRUE while homing is active.
fbPower[2].Power(
    Enable := TRUE,
    Enable_Positive := bHomingOverride OR fbLimSwStatus[2].LimitForwardEnable,
    Enable_Negative := bHomingOverride OR fbLimSwStatus[2].LimitBackwardEnable,
    Override := 100
);

// == State Machine ==
CASE nTestStep OF
    0: // Enable backlash compensation, but it must be suppressed when homing
        fbBacklashCompensation.EnableBacklashCompensation(UserEnable := TRUE, Compensation := 1.0);
        nTestStep := 1;
    1: // Wait for power enable before issuing home command
        IF fbPower[2].PowerIsEnabled THEN
			fbBacklashCompensation.BacklashCompensation(Enable := FALSE, RampVelo := 10.0);
            // Set override for homing
            bHomingOverride := TRUE;
            // Initiate homing sequence
			
            fbHome.Home(Position := 20.0, BufferMode := MC_Aborting);
            nTestStep := 2;
        END_IF
    2: // Wait until homing is busy (started)
        IF fbHome.Busy THEN
            AssertFalse(
                Condition := fbBacklashCompensation.Status,
                Message := 'Backlash must be disabled after homing started #2'
            );
            nTestStep := 3;
        END_IF
    3: // Simulate forward cam switch pulse for homing
        IF fbCamSwitchPulserSearch.Q THEN
            fbLimSwStatus[2].LimitForwardEnable := FALSE;
            fbCamSwitchPulserSearch.IN := FALSE;
            fbCamSwitchPulserSync.IN := TRUE;
            nTestStep := 4;
        END_IF
    4: // Simulate cam switch releasing back to TRUE
        IF fbCamSwitchPulserSync.Q THEN
            fbLimSwStatus[2].LimitForwardEnable := TRUE;
            nTestStep := 5;
        END_IF
    5: // When homing is done, stop override
        IF fbHome.Done THEN
            bHomingOverride := FALSE;
            nTestStep := 6;
        END_IF
END_CASE

// -- Cyclic calls to all dependencies --
fbAxisRef[2].ReadStatus();
fbBacklashCompensation();
fbHome();
fbCamSwitchPulserSearch();
fbCamSwitchPulserSync();
fbTestTimer();

// -- Assertion and test finish --
IF nTestStep = 6 THEN
    AssertTrue(
        Condition := (fbAxisRef[2].NcToPlc.ActPos - fbAxisRef[2].NcToPlc.ActPosWithoutPosCorrection) = 0,
        Message := 'Backlash compensation must be enabled #3'
    );
    TEST_FINISHED();

ELSIF fbTestTimer.Q THEN
    AssertTrue(
        Condition := FALSE,
        Message := CONCAT('Timed out at step: ', TO_STRING(nTestStep))
    );
    TEST_FINISHED();
END_IF
END_METHOD

METHOD PRIVATE GivenHomeCmdHomeViaHighModeAndHomeSwPulseThenMoveToUserDefineOffset_Test3
VAR_INST
    fbHome : FB_HomeNC(
		AxisRef:=fbAxisRef[3],
		iLimSwStatus:=fbLimSwStatus[3],
		iMotionLogger:=fbMotionLogger[3]
	) := ( Mode:=E_EpicsHomeCmd.HOME_VIA_HIGH );
	
    fbTestTimer: TON := (IN:=TRUE, PT:=T#5S);
    fbCamSwitchPulserSearch: TON := (IN:=TRUE, PT:=T#500MS);
    fbCamSwitchPulserSync: TON := (PT:=T#1000MS);
    nTestStep : INT;
    fExpectedPosition : LREAL := 20.0;
    fActPosition : LREAL;
    bCalibrated: BOOL;
    // reset this when error or homeDone
    bHomingOverride : BOOL := TRUE;

END_VAR
TEST(__POUNAME());

// Cyclic block calls
fbLimSwStatus[3]();
fbMotionLogger[3]();

fbPower[3].Power(
    Enable := TRUE,
    Enable_Positive := bHomingOverride OR fbLimSwStatus[3].LimitForwardEnable,
    Enable_Negative := bHomingOverride OR fbLimSwStatus[3].LimitBackwardEnable,
    Override := 100.0
);

CASE nTestStep OF
    0:
        IF fbPower[3].PowerIsEnabled THEN
            // Initiate Home command when power is ready
            fbHome.Home(Position := fExpectedPosition, BufferMode := MC_BufferMode.MC_Aborting);
            nTestStep := 1;
        END_IF
    1:
        // Simulate forward cam switch pulse for homing
        IF fbCamSwitchPulserSearch.Q THEN
            fbLimSwStatus[3].LimitHome := TRUE;
            fbCamSwitchPulserSearch.IN := FALSE;
            fbCamSwitchPulserSync.IN := TRUE;
            nTestStep := 2;
        END_IF
    2:
        // Clear home limit after sync pulse
        IF fbCamSwitchPulserSync.Q THEN
            fbLimSwStatus[3].LimitHome := FALSE;
            nTestStep := 3;
        END_IF
    3:
        // Wait for the home sequence to finish
        IF fbHome.Done THEN
            nTestStep := 4;
        END_IF
END_CASE

// Cyclic calls
fbAxisRef[3].ReadStatus();
fbPower[3]();
fbHome();
fbCamSwitchPulserSearch();
fbCamSwitchPulserSync();
fbTestTimer();

IF nTestStep = 4 THEN
    bCalibrated := fbHome.Done;
    AssertEquals_BOOL(
        Expected := TRUE,
        Actual := fbAxisRef[3].Status.Homed,
        Message := 'Axis not calibrated #1'
    );
    AssertEquals_LREAL(
        Delta := 0.001,
        Expected := fExpectedPosition,
        Actual := fbAxisRef[3].NcToPlc.ActPos,
        Message := 'Position is not the expected #2'
    );
    TEST_FINISHED();

ELSIF fbTestTimer.Q THEN
    AssertTrue(
        Condition := FALSE,
        Message := CONCAT('Timed out at step: ', TO_STRING(nTestStep))
    );
    TEST_FINISHED();
END_IF
END_METHOD

METHOD PRIVATE GivenHomeCmdHomeViaHighModeForwardSwPulseBeforeHomeSwPulseThenMoveToUserDefineOffset_Test4
VAR_INST
    fbHome : FB_HomeNC(
		AxisRef:=fbAxisRef[4],
		iLimSwStatus:=fbLimSwStatus[4],
		iMotionLogger:=fbMotionLogger[4]
	) := ( Mode := E_EpicsHomeCmd.HOME_VIA_HIGH );
	
    fbTestTimer: TON := (IN:=TRUE, PT:=T#5S);
    fbCamSwitchPulserSearch: TON := (IN:=TRUE, PT:=T#500MS);
    fbCamSwitchPulserSync: TON := (PT:=T#1000MS);
    nTestStep : INT;
    fExpectedPosition : LREAL := 20.0;
    fActPosition : LREAL;
    bCalibrated: BOOL;
    // reset this when error or homeDone
    bHomingOverride : BOOL := TRUE;
END_VAR
TEST(__POUNAME());

// Cyclic preparation and block invocation
fbAxisRef[4].ReadStatus();
fbLimSwStatus[4]();
fbMotionLogger[4]();
fbPower[4].Power(
    Enable := TRUE,
    Enable_Positive := bHomingOverride OR fbLimSwStatus[4].LimitForwardEnable,
    Enable_Negative := bHomingOverride OR fbLimSwStatus[4].LimitForwardEnable, // Note: both positive and negative use ForwardEnable here
    Override := 100.0
);

// Stepwise homing process
CASE nTestStep OF
    0: // Await full power-up, start first stage home
        IF fbPower[4].PowerIsEnabled THEN
            fbHome.Home(Position := fExpectedPosition, BufferMode := MC_BufferMode.MC_Aborting);
            nTestStep := 1;
        END_IF
    1: // Simulate Forward Limit pulse (stage 1 complete)
        IF fbCamSwitchPulserSearch.Q THEN
            fbLimSwStatus[4].LimitForwardEnable := FALSE;
            fbCamSwitchPulserSearch.IN := FALSE;
            fbCamSwitchPulserSync.IN := TRUE;
            nTestStep := 2;
        END_IF
    2: // Release Forward Limit (simulate rising edge)
        IF fbCamSwitchPulserSync.Q THEN
            fbLimSwStatus[4].LimitForwardEnable := TRUE;
            nTestStep := 3;
        END_IF
    3: // When forward limit home is done, prepare for the home switch
        IF fbHome.LimHomeDone THEN
            fbCamSwitchPulserSearch.IN := TRUE;
            fbCamSwitchPulserSync.IN := FALSE;
            nTestStep := 4;
        END_IF
    4: // Simulate Home switch pulse
        IF fbCamSwitchPulserSearch.Q THEN
            fbLimSwStatus[4].LimitHome := TRUE;
            fbCamSwitchPulserSearch.IN := FALSE;
            fbCamSwitchPulserSync.IN := TRUE;
            nTestStep := 5;
        END_IF
    5: // Release Home switch
        IF fbCamSwitchPulserSync.Q THEN
            fbLimSwStatus[4].LimitHome := FALSE;
            nTestStep := 6;
        END_IF
    6: // Wait for homing full completion
        IF fbHome.Done THEN
            nTestStep := 7;
        END_IF
END_CASE

// Cyclic calls required for simulation and status updates
fbPower[4]();
fbHome();
fbCamSwitchPulserSearch();
fbCamSwitchPulserSync();
fbTestTimer();

// Finish test if homing is complete (step 7), or timeout
IF nTestStep = 7 THEN
    bCalibrated := fbHome.Done;
    AssertEquals_BOOL(
        Expected := TRUE,
        Actual := fbAxisRef[4].Status.Homed,
        Message := 'Axis not calibrated #1'
    );
    AssertEquals_LREAL(
        Delta := 0.001,
        Expected := fExpectedPosition,
        Actual := fbAxisRef[4].NcToPlc.ActPos,
        Message := 'Position is not the expected #2'
    );
    TEST_FINISHED();

ELSIF fbTestTimer.Q THEN
    AssertTrue(
        Condition := FALSE,
        Message := CONCAT('Timed out at step: ', TO_STRING(nTestStep))
    );
    TEST_FINISHED();
END_IF
END_METHOD

METHOD PRIVATE GivenHomeCmdHomeViaLowModeAndHomeSwPulseThenMoveToUserDefineOffset_Test5
VAR_INST
    fbHome : FB_HomeNC(
		AxisRef:=fbAxisRef[5],
		iLimSwStatus:=fbLimSwStatus[5],
		iMotionLogger:=fbMotionLogger[5]
	) := ( Mode := E_EpicsHomeCmd.HOME_VIA_LOW );
	
    fbTestTimer: TON := (IN:=TRUE, PT:=T#5S);
    fbCamSwitchPulserSearch: TON := (IN:=TRUE, PT:=T#500MS);
    fbCamSwitchPulserSync: TON := (PT:=T#1000MS);
    nTestStep : INT;
    fExpectedPosition : LREAL := 20.0;
    fActPosition : LREAL;
	bCalibrated: BOOL;
    // reset this when error or homeDone
    bHomingOverride : BOOL := TRUE;

END_VAR
TEST(__POUNAME());

// Cyclic status/logic blocks
fbLimSwStatus[5]();
fbMotionLogger[5]();

fbPower[5].Power(
    Enable := TRUE,
    Enable_Positive := bHomingOverride OR fbLimSwStatus[5].LimitForwardEnable,
    Enable_Negative := bHomingOverride OR fbLimSwStatus[5].LimitBackwardEnable,
    Override := 100.0
);

// State machine for homing by home switch
CASE nTestStep OF
    0: // Wait for power to enable before starting home sequence
        IF fbPower[5].PowerIsEnabled THEN
            fbHome.Home(Position := fExpectedPosition, BufferMode := MC_BufferMode.MC_Aborting);
            nTestStep := 1;
        END_IF
    1: // Simulate cam switch pulse: set home limit
        IF fbCamSwitchPulserSearch.Q THEN
            fbLimSwStatus[5].LimitHome := TRUE;
            fbCamSwitchPulserSearch.IN := FALSE;
            fbCamSwitchPulserSync.IN := TRUE;
            nTestStep := 2;
        END_IF
    2: // Simulate sync pulse: clear home limit
        IF fbCamSwitchPulserSync.Q THEN
            fbLimSwStatus[5].LimitHome := FALSE;
            nTestStep := 3;
        END_IF
    3: // Wait for homing to complete
        IF fbHome.Done THEN
            nTestStep := 4;
        END_IF
    4:
        // No actions; test finishes in the assertion below
END_CASE

// Always cycle these for PLC logic to work
fbAxisRef[5].ReadStatus();
fbPower[5]();
fbHome();
fbCamSwitchPulserSearch();
fbCamSwitchPulserSync();
fbTestTimer();

// Assertions and test finish
IF nTestStep = 4 THEN
    bCalibrated := fbHome.Done;
    AssertEquals_BOOL(
        Expected := TRUE,
        Actual := fbAxisRef[5].Status.Homed,
        Message := 'Axis not calibrated #1'
    );
    AssertEquals_LREAL(
        Delta := 0.001,
        Expected := fExpectedPosition,
        Actual := fbAxisRef[5].NcToPlc.ActPos,
        Message := 'Position is not the expected #2'
    );
    TEST_FINISHED();

ELSIF fbTestTimer.Q THEN
    AssertTrue(
        Condition := FALSE,
        Message := CONCAT('Timed out at step: ', TO_STRING(nTestStep))
    );
    TEST_FINISHED();
END_IF
END_METHOD

METHOD PRIVATE GivenHomeCmdHomeViaLowModeBackwardSwPulseBeforeHomeSwPulseThenMoveToUserDefineOffset_Test6
VAR_INST
    fbHome : FB_HomeNC(
		AxisRef:=fbAxisRef[6],
		iLimSwStatus:=fbLimSwStatus[6],
		iMotionLogger:=fbMotionLogger[6]
	) := ( Mode:= E_EpicsHomeCmd.HOME_VIA_LOW );
	
    fbTestTimer: TON := (IN:=TRUE, PT:=T#5S);
    fbCamSwitchPulserSearch: TON := (IN:=TRUE, PT:=T#500MS);
    fbCamSwitchPulserSync: TON := (PT:=T#1000MS);
    nTestStep : INT;
    fExpectedPosition : LREAL := 20.0;
    fActPosition : LREAL;
	bCalibrated: BOOL;
    // reset this when error or homeDone
    bHomingOverride : BOOL := TRUE;

END_VAR
TEST(__POUNAME());

// Always call these each cycle for correct PLC scan semantics
fbAxisRef[6].ReadStatus();
fbLimSwStatus[6]();
fbMotionLogger[6]();

fbPower[6].Power(
    Enable := TRUE,
    Enable_Positive := bHomingOverride OR fbLimSwStatus[6].LimitForwardEnable,
    Enable_Negative := bHomingOverride OR fbLimSwStatus[6].LimitBackwardEnable,
    Override := 100.0
);

// State machine for negative (backward) limit then home
CASE nTestStep OF
    0: // Wait for power ready, then start home
        IF fbPower[6].PowerIsEnabled THEN
            fbHome.Home(Position := fExpectedPosition, BufferMode := MC_BufferMode.MC_Aborting);
            nTestStep := 1;
        END_IF

    1: // Simulate cam pulse: deactivate backward limit
        IF fbCamSwitchPulserSearch.Q THEN
            fbLimSwStatus[6].LimitBackwardEnable := FALSE;
            fbCamSwitchPulserSearch.IN := FALSE;
            fbCamSwitchPulserSync.IN := TRUE;
            nTestStep := 2;
        END_IF

    2: // Reactivate backward limit on sync pulse
        IF fbCamSwitchPulserSync.Q THEN
            fbLimSwStatus[6].LimitBackwardEnable := TRUE;
            nTestStep := 3;
        END_IF

    3: // Wait for negative-limit home done, then prep second stage (home switch)
        IF fbHome.LimHomeDone THEN
            fbCamSwitchPulserSearch.IN := TRUE;
            fbCamSwitchPulserSync.IN := FALSE;
            nTestStep := 4;
        END_IF

    4: // Simulate home switch pulse
        IF fbCamSwitchPulserSearch.Q THEN
            fbLimSwStatus[6].LimitHome := TRUE;
            fbCamSwitchPulserSearch.IN := FALSE;
            fbCamSwitchPulserSync.IN := TRUE;
            nTestStep := 5;
        END_IF

    5: // Deactivate home switch after sync pulse
        IF fbCamSwitchPulserSync.Q THEN
            fbLimSwStatus[6].LimitHome := FALSE;
            nTestStep := 6;
        END_IF

    6: // Wait for full home sequence completion
        IF fbHome.Done THEN
            nTestStep := 7;
        END_IF

    7: // Test ends — handled below
END_CASE

// Cyclic calls
fbPower[6]();
fbHome();
fbCamSwitchPulserSearch();
fbCamSwitchPulserSync();
fbTestTimer();

// Assertion and finish logic
IF nTestStep = 7 THEN
    bCalibrated := fbHome.Done;

    AssertEquals_BOOL(
        Expected := TRUE,
        Actual := fbAxisRef[6].Status.Homed,
        Message := 'Axis not calibrated #1'
    );

    AssertEquals_LREAL(
        Delta := 0.001,
        Expected := fExpectedPosition,
        Actual := fbAxisRef[6].NcToPlc.ActPos,
        Message := 'Position is not the expected #2'
    );

    TEST_FINISHED();

ELSIF fbTestTimer.Q THEN
    AssertTrue(
        Condition := FALSE,
        Message := CONCAT('Timed out at step: ', TO_STRING(nTestStep))
    );
    TEST_FINISHED();
END_IF
END_METHOD

METHOD PRIVATE GivenHomeCmdLowLimitModeAndABackwardSwPulseThenHomeDoneAndPositionSetToUserDefineOffset_Test7
VAR_INST
    fbHome : FB_HomeNC(
		AxisRef:=fbAxisRef[7],
		iLimSwStatus:=fbLimSwStatus[7],
		iMotionLogger:=fbMotionLogger[7]
	) := ( Mode:= E_EpicsHomeCmd.LOW_LIMIT );
    fbTestTimer: TON := (IN:=TRUE, PT:=T#5S);
    fbCamSwitchPulserSearch: TON := (IN:=TRUE, PT:=T#500MS);
    fbCamSwitchPulserSync: TON := (PT:=T#1000MS);
    nTestStep : INT;
    fExpectedPosition : LREAL := 20.0;
    fActPosition : LREAL;
    bCalibrated: BOOL;
    // reset this when error or homeDone
    bHomingOverride : BOOL := TRUE;
END_VAR
TEST(__POUNAME());

// Cyclically called blocks
fbLimSwStatus[7]();
fbMotionLogger[7]();

fbPower[7].Power(
    Enable := TRUE,
    Enable_Positive := bHomingOverride OR fbLimSwStatus[7].LimitForwardEnable,
    Enable_Negative := bHomingOverride OR fbLimSwStatus[7].LimitBackwardEnable,
    Override := 100.0
);

// State machine for negative (backward) limit homing
CASE nTestStep OF
    0: // Wait for power enabled, then start homing
        IF fbPower[7].PowerIsEnabled THEN
            fbHome.Home(Position := fExpectedPosition, BufferMode := MC_BufferMode.MC_Aborting);
            nTestStep := 1;
        END_IF

    1: // Simulate cam pulse to release backward limit
        IF fbCamSwitchPulserSearch.Q THEN
            fbLimSwStatus[7].LimitBackwardEnable := FALSE;
            fbCamSwitchPulserSearch.IN := FALSE;
            fbCamSwitchPulserSync.IN := TRUE;
            nTestStep := 2;
        END_IF

    2: // Simulate restoring backward limit
        IF fbCamSwitchPulserSync.Q THEN
            fbLimSwStatus[7].LimitBackwardEnable := TRUE;
            nTestStep := 3;
        END_IF

    3: // Wait for homing to complete
        IF fbHome.Done THEN
            nTestStep := 4;
        END_IF

    4: // Test ends; assertions below
END_CASE

// Always cycle axis status, home FB, cam pulsers, and timer
fbAxisRef[7].ReadStatus();
fbHome();
fbCamSwitchPulserSearch();
fbCamSwitchPulserSync();
fbTestTimer();

// Assertion and finish
IF nTestStep = 4 THEN
    bCalibrated := fbHome.Done;
    AssertEquals_BOOL(
        Expected := TRUE,
        Actual := fbAxisRef[7].Status.Homed,
        Message := 'Axis not calibrated #1'
    );
    AssertEquals_LREAL(
        Delta := 0.001,
        Expected := fExpectedPosition,
        Actual := fbAxisRef[7].NcToPlc.ActPos,
        Message := 'Position is not the expected #2'
    );
    TEST_FINISHED();

ELSIF fbTestTimer.Q THEN
    AssertTrue(
        Condition := FALSE,
        Message := CONCAT('Timed out at step: ', TO_STRING(nTestStep))
    );
    TEST_FINISHED();
END_IF
END_METHOD

METHOD PRIVATE GivenHomeCmdNoneModeThenSetHomeFlag_Test8
VAR_INST
    fbHome : FB_HomeNC(
		AxisRef:=fbAxisRef[8],
		iLimSwStatus:=fbLimSwStatus[8],
		iMotionLogger:=fbMotionLogger[8]
	):=(Mode:=E_EpicsHomeCmd.NONE);
    fbTestTimer: TON := (IN:=TRUE, PT:=T#5S);
    nTestStep : INT;
END_VAR
TEST(__POUNAME());

// Always call these each scan
fbLimSwStatus[8]();
fbMotionLogger[8]();

// State machine for basic home sequence
CASE nTestStep OF
    0: // Enable axis power
        fbPower[8].Power(
            Enable := TRUE,
            Enable_Positive := fbLimSwStatus[8].LimitForwardEnable,
            Enable_Negative := fbLimSwStatus[8].LimitBackwardEnable,
            Override := 100.0
        );
        nTestStep := 1;

    1: // Wait for power to come up, then issue Home command
        IF fbPower[8].PowerIsEnabled THEN
            fbHome.Home(Position := 0.0, BufferMode := MC_BufferMode.MC_Aborting);
            nTestStep := 2;
        END_IF

    2: // Wait for homing to finish
        IF fbHome.Done THEN
            nTestStep := 3;
        END_IF

    3: // Test ends; assertion and finish below
END_CASE

// Required cyclic calls
fbPower[8]();
fbHome();
fbTestTimer(IN := TRUE);

// Assertion & finish logic
IF nTestStep = 3 THEN
    // You may add validation here (homed position, calibrated flag, etc.) if required
    TEST_FINISHED();
ELSIF fbTestTimer.Q THEN
    AssertTrue(
        Condition := FALSE,
        Message := CONCAT('Timed out at step: ', TO_STRING(nTestStep))
    );
    TEST_FINISHED();
END_IF
END_METHOD

METHOD PRIVATE GivenHomeCmdSetToHighLimitAndHighLimitPulseThenSetHomeDoneAndPositionToUserDefineOffset_Test9
VAR_INST
    fbHome : FB_HomeNC(
		AxisRef:=fbAxisRef[9],
		iLimSwStatus:=fbLimSwStatus[9],
		iMotionLogger:=fbMotionLogger[9]
	):=(Mode:=E_EpicsHomeCmd.HIGH_LIMIT);
	
    fbTestTimer: TON := (IN:=TRUE, PT:=T#5S);
    fbCamSwitchPulserSearch: TON := (IN:=TRUE, PT:=T#500MS);
    fbCamSwitchPulserSync: TON := (PT:=T#1000MS);
    nTestStep : INT;
    fExpectedPosition : LREAL := 20.0;
    fActPosition : LREAL;
    bCalibrated: BOOL;
    // reset this when error or homeDone
    bHomingOverride : BOOL := TRUE;
END_VAR
TEST(__POUNAME());

// Cyclic calls: always invoked every scan
fbLimSwStatus[9]();
fbMotionLogger[9]();
fbPower[9].Power(
    Enable := TRUE,
    Enable_Positive := bHomingOverride OR fbLimSwStatus[9].LimitForwardEnable,
    Enable_Negative := bHomingOverride OR fbLimSwStatus[9].LimitBackwardEnable,
    Override := 100.0
);

// Homing state machine
CASE nTestStep OF
    0: // Wait for power enabled, then start homing command
        IF fbPower[9].PowerIsEnabled THEN
            fbHome.Home(Position := fExpectedPosition, BufferMode := MC_BufferMode.MC_Aborting);
            nTestStep := 1;
        END_IF

    1: // Simulate cam pulse to clear forward limit
        IF fbCamSwitchPulserSearch.Q THEN
            fbLimSwStatus[9].LimitForwardEnable := FALSE;
            fbCamSwitchPulserSearch.IN := FALSE;
            fbCamSwitchPulserSync.IN := TRUE;
            nTestStep := 2;
        END_IF

    2: // Simulate restoring forward limit
        IF fbCamSwitchPulserSync.Q THEN
            fbLimSwStatus[9].LimitForwardEnable := TRUE;
            nTestStep := 3;
        END_IF

    3: // Wait for homing to complete
        IF fbHome.Done THEN
            nTestStep := 4;
        END_IF

    4: // Test ends, assertions handled below
END_CASE

// Always called each scan
fbAxisRef[9].ReadStatus();
fbHome();
fbCamSwitchPulserSearch();
fbCamSwitchPulserSync();
fbTestTimer();

// Assertion and finish
IF nTestStep = 4 THEN
    bCalibrated := fbHome.Done;
    AssertEquals_BOOL(
        Expected := TRUE,
        Actual := fbAxisRef[9].Status.Homed,
        Message := 'Axis not calibrated #1'
    );
    AssertEquals_LREAL(
        Delta := 0.001,
        Expected := fExpectedPosition,
        Actual := fbAxisRef[9].NcToPlc.ActPos,
        Message := 'Position is not the expected #2'
    );
    TEST_FINISHED();

ELSIF fbTestTimer.Q THEN
    AssertTrue(
        Condition := FALSE,
        Message := CONCAT('Timed out at step: ', TO_STRING(nTestStep))
    );
    TEST_FINISHED();
END_IF
END_METHOD

METHOD PRIVATE GivenMoveCmdNegativeBacklashCompensationActiveThenReverseMoveIsCompensated_Test10
VAR_INST
    // Subjects under tests
    fbBacklashCompensation : FB_BacklashCompensationNC(AxisRef := fbAxisRef[10],  iMotionLogger:= fbMotionLogger[10]);
    fbMoveAbsolute : FB_MoveAbsoluteNC(AxisRef := fbAxisRef[10],  iMotionLogger:= fbMotionLogger[10]);
    // Backalsh is testing on simulated NC axis in Homing and PTP
    fbTestTimer : TON := (PT := T#5S, IN := TRUE);
    nTestStep : INT;;

END_VAR
TEST(__POUNAME());

// Must be called cyclically
fbPower[10].Power(
    Enable := TRUE,
    Enable_Positive := fbLimSwStatus[10].LimitForwardEnable,
    Enable_Negative := fbLimSwStatus[10].LimitBackwardEnable,
    Override := 100
);

CASE nTestStep OF
    // Enable compensation, but status should still be OFF initially
    0:
        fbBacklashCompensation.EnableBacklashCompensation(UserEnable := TRUE, Compensation := -4.0);
        nTestStep := 1;
	1:
		fbBacklashCompensation.BacklashCompensation(Enable := TRUE, RampVelo := 10.0);
		nTestStep := 2;
    2:
        AssertTrue(
            Condition := fbBacklashCompensation.Status,
            Message := 'Backlash compensation must be enabled #2'
        );
        nTestStep := 3;

    // Start negative move (direction should not apply backlash compensation here)
    3:
        IF fbPower[10].PowerIsEnabled THEN
            fbMoveAbsolute.MoveAbsolute(
                Position := -10.0,
                Velocity := 100,
                Acceleration := 200,
                Deceleration := 200
            );
            nTestStep := 4;
        END_IF

    // Assert compensation does not apply after negative move
   4:
        IF fbMoveAbsolute.Done THEN
            AssertTrue(
                Condition := (fbAxisRef[10].NcToPlc.ActPos - fbAxisRef[10].NcToPlc.ActPosWithoutPosCorrection) = 0,
                Message := 'No Backlash compensation in this direction #3'
            );
            nTestStep := 5;
        END_IF

    // Start reverse move (should apply backlash compensation)
   5:
        fbMoveAbsolute.MoveAbsolute(
            Position := 20.0,
            Velocity := 100,
            Acceleration := 200,
            Deceleration := 200
        );
        nTestStep := 6;

    // Assert compensation is applied after reverse move
   6:
        IF fbMoveAbsolute.Done THEN
            AssertTrue(
                Condition := (fbAxisRef[10].NcToPlc.ActPos - fbAxisRef[10].NcToPlc.ActPosWithoutPosCorrection) = 4,
                Message := 'Current backlash must be 4 #4'
            );
            nTestStep := 7;
        END_IF

END_CASE

// Required cyclic calls
fbBacklashCompensation();
fbMoveAbsolute();
fbTestTimer();

// Final assertion and finish
IF nTestStep = 7 THEN
    AssertTrue(
        Condition := fbBacklashCompensation.Status,
        Message := 'Backlash compensation must stay enabled after absolute move #5'
    );
    TEST_FINISHED();

ELSIF fbTestTimer.Q THEN
    AssertTrue(
        Condition := FALSE,
        Message := CONCAT('Timed out at step: ', TO_STRING(nTestStep))
    );
    TEST_FINISHED();
END_IF
END_METHOD

METHOD PRIVATE GivenMoveCmdPositiveBacklashCompensationActiveThenReverseMoveIsCompensated_Test11
VAR_INST
    // Subjects under test
    fbBacklashCompensation : FB_BacklashCompensationNC(AxisRef := fbAxisRef[11],  iMotionLogger:= fbMotionLogger[11]);
	fbMoveAbsolute : FB_MoveAbsoluteNC(AxisRef := fbAxisRef[11],  iMotionLogger:= fbMotionLogger[11]);
    // Backalsh is testing on simulated NC axis in Homing and PTP
    fbTestTimer : TON := (PT := T#5S, IN := TRUE);
    nTestStep : INT;

    


END_VAR
TEST(__POUNAME());

// Must be called cyclically
fbPower[11].Power(
    Enable := TRUE,
    Enable_Positive := fbLimSwStatus[11].LimitForwardEnable,
    Enable_Negative := fbLimSwStatus[11].LimitBackwardEnable,
    Override := 100
);

CASE nTestStep OF
    // Enable compensation, but status should still be OFF initially
    0:
        fbBacklashCompensation.EnableBacklashCompensation(UserEnable := TRUE, Compensation := 4.0);
        nTestStep := 1;
	1:
		fbBacklashCompensation.BacklashCompensation(Enable := TRUE, RampVelo := 10.0);
		nTestStep := 2;
    2:
        AssertTrue(
            Condition := fbBacklashCompensation.Status,
            Message := 'Backlash compensation must be enabled #2'
        );
        nTestStep := 3;

    // Start negative move (direction should not apply backlash compensation here)
    3:
        IF fbPower[11].PowerIsEnabled THEN
            fbMoveAbsolute.MoveAbsolute(
                Position :=50.0,
                Velocity := 100,
                Acceleration := 200,
                Deceleration := 200
            );
            nTestStep := 4;
        END_IF

    // Assert compensation does not apply after negative move
   4:
        IF fbMoveAbsolute.Done THEN
            AssertTrue(
                Condition := (fbAxisRef[11].NcToPlc.ActPos - fbAxisRef[11].NcToPlc.ActPosWithoutPosCorrection) = 0,
                Message := 'No Backlash compensation in this direction #3'
            );
            nTestStep := 5;
        END_IF

    // Start reverse move (should apply backlash compensation)
   5:
        fbMoveAbsolute.MoveAbsolute(
            Position := 25.0,
            Velocity := 100,
            Acceleration := 200,
            Deceleration := 200
        );
        nTestStep := 6;

    // Assert compensation is applied after reverse move
   6:
        IF fbMoveAbsolute.Done THEN
            AssertTrue(
                Condition := (fbAxisRef[11].NcToPlc.ActPos - fbAxisRef[11].NcToPlc.ActPosWithoutPosCorrection) = 4,
                Message := 'Current backlash must be 4 #4'
            );
            nTestStep := 7;
        END_IF

END_CASE

// Required cyclic calls
fbBacklashCompensation();
fbMoveAbsolute();
fbTestTimer();

// Final assertion and finish
IF nTestStep = 7 THEN
    AssertTrue(
        Condition := fbBacklashCompensation.Status,
        Message := 'Backlash compensation must stay enabled after absolute move #5'
    );
    TEST_FINISHED();

ELSIF fbTestTimer.Q THEN
    AssertTrue(
        Condition := FALSE,
        Message := CONCAT('Timed out at step: ', TO_STRING(nTestStep))
    );
    TEST_FINISHED();
END_IF
END_METHOD

METHOD PRIVATE GivenPowerIsEnabledAbsoluteMoveIfResetThenMoveIsAbortedAndResetDoneIsRetained_Test16
VAR_INST
    // Subjects under test
    fbMoveAbsolute : FB_MoveAbsoluteNC(AxisRef := fbAxisRef[16], iMotionLogger:= fbMotionLogger[16]);
    fbReset : FB_ResetNC(AxisRef := fbAxisRef[16], iMotionLogger:= fbMotionLogger[16]);
    fbTestTimer : TON := (PT := T#3S, IN := TRUE);
    fbInMotionTimer : TON := (PT := T#1S, IN := FALSE);
    nTestStateStep : INT;
END_VAR
TEST(__POUNAME());

// Cyclic power logic
fbPower[16].Power(
    Enable := TRUE,
    Enable_Positive := fbLimSwStatus[16].LimitForwardEnable,
    Enable_Negative := fbLimSwStatus[16].LimitBackwardEnable,
    Override := 100
);

// State machine for move + reset abort
CASE nTestStateStep OF
    0: // Wait for axis power before starting move
        IF fbPower[16].PowerIsEnabled THEN
            nTestStateStep := 1;
        END_IF

    1: // Issue move absolute
        fbMoveAbsolute.MoveAbsolute(
            Position := 100,
            Velocity := 100,
            Acceleration := 50,
            Deceleration := 50
        );
        nTestStateStep := 2;

    2: // Wait for axis to become busy; start timer
        IF fbMoveAbsolute.Busy THEN
            fbInMotionTimer.IN := TRUE;
            nTestStateStep := 3;
        END_IF

    3: // When timer elapses, send Reset to abort move
        IF fbInMotionTimer.Q THEN
            fbReset.Reset();
            fbInMotionTimer.IN := FALSE;
            nTestStateStep := 4;
        END_IF

    4: // Wait for reset to be done (move abort completion)
        IF fbReset.Done THEN
            nTestStateStep := 5;
        END_IF
END_CASE

// Cyclic calls for status and timers
fbInMotionTimer();
fbAxisRef[16].ReadStatus();
fbMoveAbsolute();
fbReset();
fbTestTimer();

// Assertion and finish logic
IF nTestStateStep = 5 THEN
    AssertTrue(
        Condition := fbMoveAbsolute.Aborted,
        Message := 'Expected CommandAborted'
    );
    AssertTrue(
        Condition := fbReset.Done,
        Message := 'Expected Reset.Done'
    );
    AssertFalse(
        Condition := fbReset.Busy,
        Message := 'Expected Reset not busy'
    );
    TEST_FINISHED();

ELSIF fbTestTimer.Q THEN
    AssertTrue(
        Condition := FALSE,
        Message := CONCAT('Timed out at step: ', TO_STRING(nTestStateStep))
    );
    TEST_FINISHED();
END_IF
END_METHOD

METHOD PRIVATE GivenPowerIsEnabledAndAbsoluteMoveStartedIfHaltSignalThenMoveIsAbortedAndHaltDoneIsRetained_Test15
VAR_INST
    // Subjects under test
    fbMoveAbsolute : FB_MoveAbsoluteNC(AxisRef := fbAxisRef[15], iMotionLogger:= fbMotionLogger[15]);
    fbHalt : FB_HaltNC(AxisRef := fbAxisRef[15], iMotionLogger:= fbMotionLogger[15]);
    fbTestTimer : TON := (PT := T#3S, IN := TRUE);
    fbInMotionTimer : TON := (PT := T#1S, IN := FALSE);
    nTestStateStep : INT;;
END_VAR
TEST(__POUNAME());

// Always called per scan
fbPower[15].Power(
    Enable := TRUE,
    Enable_Positive := fbLimSwStatus[15].LimitForwardEnable,
    Enable_Negative := fbLimSwStatus[15].LimitBackwardEnable,
    Override := 100
);

// State machine for move + halt
CASE nTestStateStep OF
    0 : // Wait for power-up before starting move
        IF fbPower[15].PowerIsEnabled THEN
            nTestStateStep := 1;
        END_IF

    1 : // Start move
        fbMoveAbsolute.MoveAbsolute(
            Position := 100,
            Velocity := 100,
            Acceleration := 50,
            Deceleration := 50
        );
        nTestStateStep := 2;

    2 : // Wait until move system is busy, then start in-motion timer
        IF fbMoveAbsolute.Busy THEN
            fbInMotionTimer.IN := TRUE;
            nTestStateStep := 3;
        END_IF

    3 : // When timer triggers, send Halt
        IF fbInMotionTimer.Q THEN
            fbHalt.Halt(
                Deceleration := 100,
                Jerk := 0
            );
            fbInMotionTimer.IN := FALSE;
            nTestStateStep := 4;
        END_IF

    4 : // Wait for halt done (move abort confirmation)
        IF fbHalt.Done THEN
            nTestStateStep := 5;
        END_IF

    5 : // Test ends; assertions below
        // (do nothing)
END_CASE

// Cyclic calls
fbTestTimer();
fbInMotionTimer();
fbAxisRef[15].ReadStatus();
fbMoveAbsolute();
fbHalt();

// Test result and finish logic
IF nTestStateStep = 5 THEN
    AssertTrue(
        Condition := fbMoveAbsolute.Aborted,
        Message := 'Expected CommandAborted'
    );
    AssertTrue(
        Condition := fbHalt.Done,
        Message := 'Expected Done'
    );
    AssertFalse(
        Condition := fbHalt.Busy,
        Message := 'Expected not busy'
    );
    TEST_FINISHED();

ELSIF fbTestTimer.Q THEN
    AssertTrue(
        Condition := FALSE,
        Message := CONCAT('Timed out at step: ', TO_STRING(nTestStateStep))
    );
    TEST_FINISHED();
END_IF
END_METHOD

METHOD PRIVATE GivenPowerIsEnabledAndCompletedAbsoluteMoveThenMoveAbsoluteDoneStatusRetained_Test14
VAR_INST
    fbMoveAbsolute : FB_MoveAbsoluteNC(AxisRef := fbAxisRef[14], iMotionLogger:= fbMotionLogger[14]);
    nTestStateStep : INT;
    fbTestTimer : TON := (PT := T#3S, IN := TRUE);
    fExpectedPosition: LREAL := 50.0;
END_VAR
TEST(__POUNAME());

// Always call required power block
fbPower[14].Power(
    Enable := TRUE,
    Enable_Positive := fbLimSwStatus[14].LimitForwardEnable,
    Enable_Negative := fbLimSwStatus[14].LimitBackwardEnable,
    Override := 100
);

// Stepwise state machine for the move
CASE nTestStateStep OF
    0 : // Wait for power-on before starting move
        IF fbPower[14].PowerIsEnabled THEN
            nTestStateStep := 1;
        END_IF

    1 : // Issue Move Absolute command
        fbMoveAbsolute.MoveAbsolute(
            Position := fExpectedPosition,   // Substituted value for clarity
            Velocity := 500,
            Acceleration := 1000,
            Deceleration := 1000
        );
        nTestStateStep := 2;

    2 : // Wait until move finishes
        IF fbMoveAbsolute.Done THEN
            nTestStateStep := 3;
        END_IF
END_CASE

// Cyclically called per scan
fbTestTimer();
fbAxisRef[14].ReadStatus();
fbMoveAbsolute();

// Final assertion and test finish
IF nTestStateStep = 3 THEN
    AssertEquals_LREAL(
        Delta := 0.001,
        Expected := fExpectedPosition,
        Actual := fbAxisRef[14].NcToPlc.ActPos,
        Message := 'Position is not the expected #1'
    );
    TEST_FINISHED();

ELSIF fbTestTimer.Q THEN
    AssertTrue(
        Condition := FALSE,
        Message := CONCAT('Timed out at step: ', TO_STRING(nTestStateStep))
    );
    TEST_FINISHED();
END_IF
END_METHOD

END_FUNCTION_BLOCK

// ---- POUs/FBs/NC/FB_PowerNC.TcPOU
FUNCTION_BLOCK FB_PowerNC IMPLEMENTS I_Power
VAR
    {attribute 'no_copy'}
    AxisRef : REFERENCE TO AXIS_REF;
    fbMcPower : MC_Power;
	iMotionLogger : I_MotionLogger := 0;
	rtError: R_TRIG;
END_VAR

IF NOT __ISVALIDREF(AxisRef) THEN
    RETURN;
END_IF

AxisRef.ReadStatus();

fbMcPower(
    Axis := AxisRef,
);

rtError(CLK:=fbMcPower.Error);
IF rtError.Q THEN
	iMotionLogger.Logger(Message := iMotionLogger.ErrorCodeLookup(fbMcPower.ErrorID), Level := E_MotionLogLevel.ERROR, Source := 'Power');	
END_IF

PROPERTY Busy : BOOL
GET
Busy := THIS^.fbMcPower.Busy;
END_GET
END_PROPERTY

METHOD PUBLIC CallAfterInit
VAR_INPUT
    AxisRef : REFERENCE TO AXIS_REF;
	iMotionLogger : I_MotionLogger;
END_VAR
THIS^.AxisRef REF= AxisRef;
THIS^.iMotionLogger := iMotionLogger;
END_METHOD

PROPERTY DirectionalPowerEnabled : BOOL
GET
DirectionalPowerEnabled := THIS^.fbMcPower.Enable_Negative AND THIS^.fbMcPower.Enable_Positive;
END_GET
END_PROPERTY

METHOD DisablePower
(*Use to remove power in DURING_MOTION driving mode *)
THIS^.fbMcPower(
    Axis := THIS^.AxisRef,
    Enable := FALSE
);
END_METHOD

PROPERTY Done : BOOL
GET
END_GET
END_PROPERTY

PROPERTY Error : BOOL
GET
Error := THIS^.fbMcPower.Error;
END_GET
END_PROPERTY

PROPERTY ErrorID : UDINT
GET
ErrorID := THIS^.fbMcPower.ErrorID;
END_GET
END_PROPERTY

//FB_Init is always available implicitly and it is used primarily for initialization.
//The return value is not evaluated. For a specific influence, you can also declare the
//methods explicitly and provide additional code there with the standard initialization
//code. You can evaluate the return value.
METHOD FB_Init: BOOL
VAR_INPUT
    bInitRetains: BOOL; // TRUE: the retain variables are initialized (reset warm / reset cold)
    bInCopyCode: BOOL;  // TRUE: the instance will be copied to the copy code afterward (online change)
    AxisRef : REFERENCE TO AXIS_REF;
	iMotionLogger : I_MotionLogger;
END_VAR
THIS^.AxisRef REF= AxisRef;
THIS^.iMotionLogger := iMotionLogger;
END_METHOD

PROPERTY Message : T_MAXSTRING
GET
END_GET
END_PROPERTY

PROPERTY Override : LREAL
GET
Override := THIS^.fbMcPower.Override;
END_GET
END_PROPERTY

(*When the enable flags are updated externally this must be called cyclicly*)
METHOD Power
VAR_INPUT
    Enable	: BOOL;
    Enable_Positive	: BOOL;
    Enable_Negative	: BOOL;
    Override	: LREAL := 100.0;
    BufferMode	: MC_BufferMode := MC_BufferMode.MC_Aborting;
END_VAR
(*The calling block must provide homing directional Power enables override *)
THIS^.fbMcPower(
    Axis := THIS^.AxisRef,
    Enable := Enable,
    Enable_Positive := Enable_Positive,
    Enable_Negative := Enable_Negative,
    BufferMode := BufferMode,
    Override :=Override
);
END_METHOD

PROPERTY PowerIsEnabled : BOOL
GET
PowerIsEnabled :=THIS^.fbMcPower.Status;
END_GET
END_PROPERTY

END_FUNCTION_BLOCK

// ---- POUs/FBs/NC/FB_MoveAbsoluteNC.TcPOU
FUNCTION_BLOCK FB_MoveAbsoluteNC IMPLEMENTS I_MoveAbsolute
VAR
    {attribute 'no_copy'}
    AxisRef : REFERENCE TO AXIS_REF;
    // MoveABsolute
    fbMcMoveAbsolute : MC_MoveAbsolute;
    sMessage : T_MAXSTRING;
    eMoveAbsoluteState : (WaitingMoveAbsolute, MovingAbsolute);
END_VAR

IF NOT __ISVALIDREF(THIS^.AxisRef) THEN
    RETURN;
END_IF

THIS^.AxisRef.ReadStatus();

CASE eMoveAbsoluteState OF
    WaitingMoveAbsolute :
        fbMcMoveAbsolute(
        Axis := AxisRef,
        Execute := FALSE);

    MovingAbsolute :
        fbMcMoveAbsolute(
        Axis := AxisRef,
        Execute := TRUE
        );

END_CASE

{warning 'Add property implementation'}
PROPERTY Aborted : BOOL
GET
Aborted := THIS^.fbMcMoveAbsolute.CommandAborted;
END_GET
END_PROPERTY

{warning 'Add property implementation'}
PROPERTY Active : BOOL
GET
Active := THIS^.fbMcMoveAbsolute.Active;
END_GET
END_PROPERTY

{warning 'add property implementation'}
PROPERTY Busy : BOOL
GET
Busy := THIS^.fbMcMoveAbsolute.Busy;
END_GET
END_PROPERTY

METHOD PUBLIC CallAfterInit
VAR_INPUT
    AxisRef : REFERENCE TO AXIS_REF;
END_VAR
THIS^.AxisRef REF= AxisRef;
END_METHOD

PROPERTY CommandMoveAbsolute : BOOL
SET
//bCommandMoveAbsolute := CommandMoveAbsolute;
END_SET
END_PROPERTY

{warning 'add property implementation'}
PROPERTY Done : BOOL
GET
Done := THIS^.fbMcMoveAbsolute.Done;
END_GET
END_PROPERTY

{warning 'add property implementation'}
PROPERTY Error : BOOL
GET
Error := THIS^.fbMcMoveAbsolute.Error;
END_GET
END_PROPERTY

{warning 'add property implementation'}
PROPERTY ErrorID : UDINT
GET
ErrorID := THIS^.fbMcMoveAbsolute.ErrorID;
END_GET
END_PROPERTY

METHOD FB_Init : BOOL
VAR_INPUT
    bInitRetains : BOOL; // if TRUE, the retain variables are initialized (warm start / cold start)
    bInCopyCode : BOOL;  // if TRUE, the instance afterwards gets moved into the copy code (online change)
    AxisRef : REFERENCE TO AXIS_REF;
END_VAR
THIS^.AxisRef REF= AxisRef;
END_METHOD

PROPERTY Message : T_MAXSTRING
GET
Message := sMessage;
END_GET
END_PROPERTY

METHOD MoveAbsolute
VAR_INPUT
    Position	: LREAL;
    Velocity	: LREAL;
    Acceleration	: LREAL := 0.0;
    Deceleration	: LREAL := 0.0;
    Jerk	: LREAL := 0.0;
    BufferMode	: MC_BufferMode := MC_BufferMode.MC_Aborting;
END_VAR
fbMcMoveAbsolute(Execute := FALSE,
                 Axis := THIS^.AxisRef);

fbMcMoveAbsolute(Execute := TRUE,
        Axis := THIS^.AxisRef,
    Position := Position,
    Velocity := Velocity,
    Acceleration := Acceleration,
    Deceleration := Deceleration,
    Jerk := Jerk,
    BufferMode := BufferMode);
eMoveAbsoluteState := MovingAbsolute;
END_METHOD

END_FUNCTION_BLOCK

// ---- POUs/FBs/NC/FB_HomeNC.TcPOU
FUNCTION_BLOCK FB_HomeNC IMPLEMENTS I_Home
VAR
    {attribute 'no_copy'}
    AxisRef : REFERENCE TO AXIS_REF;
    {attribute 'hide'}
    iMotionLogger : I_MotionLogger := 0;
    {attribute 'hide'}
    iLimSwStatus : I_LimSwStatus;
    fbMcHome : MC_Home;
    fbMcSetPosition : MC_SetPosition;
    fPosition : LREAL;
    fOffset : LREAL;
    {attribute 'hide'}
    nHomeState : UINT;
    //eHomeMode: E_EpicsHomeCmd :=E_EpicsHomeCmd.NONE;
    nHomeMode: INT :=E_EpicsHomeCmd.NONE;
    {attribute 'hide'}
    bForwardLimHitFirst : BOOL;
    {attribute 'hide'}
    bBackwardLimHitFirst : BOOL;
    {attribute 'hide'}
    ftForwardSwHitFirst : F_TRIG;
    {attribute 'hide'}
    ftBackwardLimHitFirst : R_TRIG;
    {attribute 'hide'}
    ftBackwardSwHitFirst: F_TRIG;
    {attribute 'hide'}
    rtHomeSwHitFirst : R_TRIG;
    {attribute 'hide'}
    bHomeSwHitFirst : BOOL;
    {attribute 'hide'}
    bHLDone : BOOL;
    {attribute 'hide'}
    rtDone : R_TRIG;
    {attribute 'hide'}
    bHomeDone: BOOL;
	rtError: R_TRIG;
	bIsLowMode : BOOL;
	bLimitEnable : BOOL;
	eInitSearchDir, eInitSyncDir, eRetrySearchDir, eRetrySyncDir : MC_Direction;
	bLimitHitFirst : BOOL;
	ftLimitHitFirst : F_TRIG; // or a reference if your F_TRIGs are function blocks per direction
	bHomeRequested: BOOL;
	bExecLatched: BOOL;
    bReadyForHome : BOOL;
    bStartHoming  : BOOL;
	eRequestedBufferMode: MC_BufferMode;
	bInterlocksOK: BOOL;
	bEdgeToStart: BOOL;
	bIsLow: BOOL;
	rtHomeRequest: R_TRIG;
	bRisingEdgeReq: BOOL;
	bAborted: BOOL;
END_VAR

// Validate reference
IF NOT __ISVALIDREF(AxisRef) THEN
    RETURN;
END_IF

// Detect the rising edge of a home request only
rtHomeRequest(CLK := bHomeRequested);
bRisingEdgeReq := rtHomeRequest.Q;

// On rising edge, check interlocks and (re)arm bStartHoming if safe
IF bRisingEdgeReq THEN
    bInterlocksOK := 
        iLimSwStatus.LimitBackwardEnable AND
        iLimSwStatus.LimitForwardEnable AND
        NOT iLimSwStatus.LimitHome;
    IF bInterlocksOK THEN
        bStartHoming := TRUE;
        //nHomeState := 0; // always reset substates for a new home request
    ELSE
        bStartHoming := FALSE;
    END_IF
END_IF

// Clear SetPosition execute, unless we just did a home (it will get set as needed)
fbMcSetPosition.Execute := FALSE;

// Prepare all parameters, substates if needed, but DO NOT call fbMcHome here!
CASE nHomeMode OF

    // -------- LOW/HIGH LIMIT (parameterized) ---------------
    E_EpicsHomeCmd.LOW_LIMIT, E_EpicsHomeCmd.HIGH_LIMIT:
        bIsLow := (nHomeMode = E_EpicsHomeCmd.LOW_LIMIT);
        fbMcHome.HomingMode             := MC_HomingMode.MC_DefaultHoming;
        fbMcHome.Options.ClearPositionLag:= TRUE;
        IF bIsLow THEN
            fbMcHome.Options.SearchDirection := MC_Direction.MC_Negative_Direction;
            fbMcHome.Options.SyncDirection   := MC_Direction.MC_Positive_Direction;
            fbMcHome.bCalibrationCam        := NOT iLimSwStatus.LimitBackwardEnable;
        ELSE
            fbMcHome.Options.SearchDirection := MC_Direction.MC_Positive_Direction;
            fbMcHome.Options.SyncDirection   := MC_Direction.MC_Negative_Direction;
            fbMcHome.bCalibrationCam        := NOT iLimSwStatus.LimitForwardEnable;
        END_IF
        // *** Only set execute ONCE (and ONCE ONLY) when MC_Home.Done is true ***
        fbMcSetPosition.Execute := fbMcHome.Done;

    // -------- HOME_VIA_LOW/HIGH (state machine) ----------
    E_EpicsHomeCmd.HOME_VIA_LOW, E_EpicsHomeCmd.HOME_VIA_HIGH:
        bIsLow := (nHomeMode = E_EpicsHomeCmd.HOME_VIA_LOW);
		fbMcHome.HomingMode := MC_HomingMode.MC_DefaultHoming;
		fbMcHome.Options.ClearPositionLag := TRUE;
        IF bIsLow THEN
            bLimitEnable := iLimSwStatus.LimitBackwardEnable;
            eInitSearchDir := MC_Direction.MC_Negative_Direction;
            eInitSyncDir := MC_Direction.MC_Positive_Direction;
            eRetrySearchDir := MC_Direction.MC_Positive_Direction;
            eRetrySyncDir := MC_Direction.MC_Negative_Direction;
            ftLimitHitFirst := ftBackwardSwHitFirst;
        ELSE
            bLimitEnable := iLimSwStatus.LimitForwardEnable;
            eInitSearchDir := MC_Direction.MC_Positive_Direction;
            eInitSyncDir := MC_Direction.MC_Negative_Direction;
            eRetrySearchDir := MC_Direction.MC_Negative_Direction;
            eRetrySyncDir := MC_Direction.MC_Positive_Direction;
            ftLimitHitFirst := ftForwardSwHitFirst;
        END_IF
        fbMcHome.bCalibrationCam := iLimSwStatus.LimitHome OR NOT bLimitEnable;

        CASE nHomeState OF
            0: // Prep initial move toward limit
                fbMcHome.Options.SearchDirection := eInitSearchDir;
                fbMcHome.Options.SyncDirection   := eInitSyncDir;
                IF fbMcHome.Busy THEN nHomeState := 1; END_IF
            1: // Arm triggers for limit/home switch events
                IF bIsLow THEN
                    ftBackwardSwHitFirst(CLK := iLimSwStatus.LimitBackwardEnable);
                ELSE
                    ftForwardSwHitFirst(CLK := iLimSwStatus.LimitForwardEnable);
                END_IF
                rtHomeSwHitFirst(CLK := iLimSwStatus.LimitHome);
                IF fbMcHome.Busy THEN
                    IF rtHomeSwHitFirst.Q THEN
                        bHomeSwHitFirst := TRUE;
                        nHomeState := 4; // home OK -- complete
                    ELSIF ftLimitHitFirst.Q THEN
                        bLimitHitFirst := TRUE;
                        nHomeState := 2; // needs retry
                    END_IF
                END_IF
            2: // Wait for MC_Home complete after hitting limit
                IF bLimitHitFirst AND fbMcHome.Done THEN
                    bHLDone := TRUE;
                    bHomeSwHitFirst := FALSE;
                    bLimitHitFirst := FALSE;
                    nHomeState := 3; // ready for retry move
                END_IF
            3: // Prep retry in opposite direction. DO NOT pulse MC_Home here!
                fbMcHome.Options.SearchDirection := eRetrySearchDir;
                fbMcHome.Options.SyncDirection := eRetrySyncDir;
                fPosition := fbMcHome.Position; // preserve/forward position if needed for MC FB
                bHomeRequested := TRUE; // re-arm the request for next scan (this pulse is handled by edge in logic above)
                bStartHoming := FALSE;  // since we just retried, need edge again next scan
                nHomeState := 4;
            4: // Wait for final MC_Home done, then MC_SetPosition
                IF fbMcHome.Done THEN
                    fbMcSetPosition.Execute := TRUE;
                    nHomeState := 5;
                END_IF
            5:
                // Latch bHomeDone below after MC_Home.Done & MC_SetPosition.Done
                IF fbMcHome.Done AND fbMcSetPosition.Done THEN
                    bHLDone := FALSE;
                    bHomeRequested := FALSE;
                    nHomeState := 6;
                END_IF
        END_CASE

    // -------- ABSOLUTE_SET ---------------
    E_EpicsHomeCmd.ABSOLUTE_SET:
        fbMcHome.HomingMode := MC_HomingMode.MC_Direct;
        fbMcHome.Options.SearchDirection := MC_Direction.MC_Undefined_Direction;
        fbMcHome.Options.SyncDirection   := MC_Direction.MC_Undefined_Direction;
        fbMcHome.Options.ClearPositionLag := TRUE;
		fbMcSetPosition.Execute := fbMcHome.Done;
    // -------- NONE (no-op) ---------------
    E_EpicsHomeCmd.NONE:
        bHomeDone := TRUE;
        bStartHoming := FALSE;
END_CASE

// --- Call MC_Home outside state machines (edge/latch logic applies to ALL states) ---
fbMcHome(
    Execute    := bStartHoming,
    Axis       := AxisRef,
    Position   := fPosition,
    BufferMode := eRequestedBufferMode
);
// (single call per scan: never call inside substates!)
// Always call MC_SetPosition for status maintenance
fbMcSetPosition(
    Axis := AxisRef,
    Mode := 0,
    Position := fPosition
);
// --- Latch 'home done' for all non-NONE modes: both MC FBs must be done ---
IF bAborted THEN
    bHomeDone := TRUE;              // Aborted home overrides
ELSE
    bHomeDone S= fbMcHome.Done AND fbMcSetPosition.Done; // Only when genuinely complete
END_IF

// Clear request as soon as MC_Home actually starts the operation
IF fbMcHome.Busy THEN
    bHomeRequested := FALSE;
END_IF

// --- Error logging ---
rtError(CLK := fbMcHome.Error OR fbMcSetPosition.Error);
IF rtError.Q AND fbMcHome.Error THEN
    iMotionLogger.Logger(
        Message := iMotionLogger.ErrorCodeLookup(fbMcHome.ErrorID),
        Level := E_MotionLogLevel.ERROR,
        Source := 'Home'
    );
ELSIF rtError.Q AND fbMcSetPosition.Error THEN
    iMotionLogger.Logger(
        Message := iMotionLogger.ErrorCodeLookup(fbMcSetPosition.ErrorID),
        Level := E_MotionLogLevel.ERROR,
        Source := 'Home'
    );
END_IF

PROPERTY Aborted : BOOL
GET
Aborted := THIS^.bAborted;
END_GET
END_PROPERTY

METHOD AbortRecovery
// Call this when you detect external halt/reset/request

// 1. Immediately stop MC_Home and MC_SetPosition
fbMcHome(
    Execute := FALSE,
    Axis    := THIS^.AxisRef
);
fbMcSetPosition(
    Execute := FALSE,
    Axis    := THIS^.AxisRef,
    Mode    := 0,
    Position:= THIS^.fPosition
);
// 2. Clear/latch all home execution state
THIS^.bHomeRequested    := FALSE;
THIS^.bExecLatched      := FALSE;
THIS^.bStartHoming      := FALSE;
THIS^.bHomeDone         := FALSE;
THIS^.bAborted          := TRUE;     
THIS^.bHLDone           := FALSE;
THIS^.bHomeSwHitFirst   := FALSE;
THIS^.bLimitHitFirst    := FALSE;

// 3. Reinitialize substates if present
THIS^.nHomeState        := 0;
END_METHOD

PROPERTY Active : BOOL
GET
Active := fbMcHome.Active;
END_GET
END_PROPERTY

PROPERTY Busy : BOOL
GET
Busy := fbMcHome.Busy;
END_GET
END_PROPERTY

METHOD PUBLIC CallAfterInit
VAR_INPUT
    AxisRef : REFERENCE TO AXIS_REF;
    iMotionLogger : I_MotionLogger;
    iLimSwStatus : I_LimSwStatus;
END_VAR
THIS^.AxisRef REF= AxisRef;
THIS^.iMotionLogger := iMotionLogger;
THIS^.iLimSwStatus:= iLimSwStatus;
END_METHOD

METHOD ClearStatus
THIS^.AbortRecovery();
// Override this as the call is a reinit one this time around.
THIS^.bAborted          := FALSE;
END_METHOD

PROPERTY Done : BOOL
GET
Done := bHomeDone;
END_GET
END_PROPERTY

PROPERTY Error : BOOL
GET
Error := fbMcHome.Error;
END_GET
END_PROPERTY

PROPERTY ErrorID : UDINT
GET
ErrorID := fbMcHome.ErrorID;
END_GET
END_PROPERTY

//FB_Init is always available implicitly and it is used primarily for initialization.
//The return value is not evaluated. For a specific influence, you can also declare the
//methods explicitly and provide additional code there with the standard initialization
//code. You can evaluate the return value.
METHOD FB_Init: BOOL
VAR_INPUT
    bInitRetains: BOOL; // TRUE: the retain variables are initialized (reset warm / reset cold)
    bInCopyCode: BOOL;  // TRUE: the instance will be copied to the copy code afterward (online change)
    AxisRef : REFERENCE TO AXIS_REF;
    iMotionLogger : I_MotionLogger;
    iLimSwStatus : I_LimSwStatus;
END_VAR
THIS^.AxisRef REF= AxisRef;
THIS^.iMotionLogger := iMotionLogger;
THIS^.iLimSwStatus:= iLimSwStatus;
END_METHOD

METHOD  Home : BOOL
VAR_INPUT
    Position        : LREAL  := DEFAULT_HOME_POSITION;
    BufferMode      : MC_BufferMode;
 	HomeMode: INT := E_EpicsHomeCmd.NONE;
END_VAR
// 1. Store input parameters for use by run()
THIS^.nHomeMode     := HomeMode;
THIS^.fPosition     := Position;
THIS^.eRequestedBufferMode   := BufferMode;

// 2. Arm the request flag for run(), and release any edge-triggered logic
THIS^.bHomeRequested := TRUE;      // "Arm" request for next scan
THIS^.bStartHoming   := FALSE;     // Ensures Execute edge happens safely in run()

// 3. Optionally, reset state/substates if using a homing substates machine
THIS^.nHomeState := 0;

// 4. Reset both MC_Home and MC_SetPosition (important for latching FBs)
fbMcHome(Execute := FALSE, Axis := THIS^.AxisRef);
fbMcSetPosition(Execute := FALSE, Axis := THIS^.AxisRef, Mode := 0, Position := Position);

// 5. Clear additional latches as needed (retry flags, home-done latch, etc.)
THIS^.bHLDone   := FALSE;
THIS^.bHomeDone   := FALSE;
THIS^.bHomeSwHitFirst := FALSE;
THIS^.bLimitHitFirst  := FALSE;
// Clear abort override for new request
THIS^.bAborted := FALSE;
// 6. Optionally, return or set OUT param if you want immediate feedback
Home := FALSE; // Will become TRUE after completion observed in run()
END_METHOD

METHOD HomeDone
fbMcHome(
	Execute := FALSE, 
	Axis := THIS^.AxisRef, 
	Done=>bHomeDone
);
END_METHOD

PROPERTY LimHomeDone : BOOL
GET
LimHomeDone := bHLDone;
END_GET
END_PROPERTY

PROPERTY Message : T_MAXSTRING
GET
END_GET
END_PROPERTY

PROPERTY Mode : INT
GET
Mode := nHomeMode;
END_GET
SET
nHomeMode := Mode;
END_SET
END_PROPERTY

PROPERTY Offset : LREAL
SET
fOffset := Offset;
END_SET
END_PROPERTY

PROPERTY Position : LREAL
SET
fPosition := Position;
END_SET
END_PROPERTY

END_FUNCTION_BLOCK

// ---- POUs/FBs/NC/FB_BacklashCompensationNC.TcPOU
FUNCTION_BLOCK FB_BacklashCompensationNC IMPLEMENTS I_BacklashCompensation
VAR_INPUT
END_VAR
VAR_OUTPUT
END_VAR
VAR
(* Other status information for users of the IOC *)
    (* Backlash compensation*)
    // Enabled axis backlash compensation
    {attribute 'pytmc' := '
        pv: PLC:bBacklashCompUserEn
        io: io
        field: ZNAM FALSE
        field: ONAM TRUE
        field: DESC Enable Backlash compensation
    '}
    bUserEnable: BOOL;

    // backlash compensation status
    {attribute 'pytmc' := '
        pv: PLC:bBacklashCompStatus
        io: i
        field: ZNAM DISABLED
        field: ONAM ENABLED
        field: DESC Backlash compensation status
    '}
    bBacklashCompStatus: BOOL;

    // Backlash compensation value
    {attribute 'pytmc' := '
        pv: PLC:fBacklashComp
        io: io
        field: DESC Backlash compensation
    '}
    fBacklashComp: LREAL := 0.0;

    // Current Backlash compensation value ?
    {attribute 'pytmc' := '
        pv: PLC:fMeasuredBacklashComp
        io: i
        field: DESC Currently applied compensation
    '}
    fActCompensation: LREAL;

    {attribute 'no_copy'}
    AxisRef : REFERENCE TO AXIS_REF;
    fbMcBacklashCompensation: MC_BacklashCompensation;
    fPrevCompensation : LREAL := 0.0;
    bActive: BOOL;
    fRampVelo : LREAL := 0.0;
    bLocalEnable : BOOL;
    bError : BOOL;
    bBusy : BOOL;
    nErrorID : UDINT;
    sMessage : T_MAXSTRING;
    eDisableMode: E_DisableMode := E_DISABLEMODE.DisableModeHold;

END_VAR

IF NOT __ISVALIDREF(THIS^.AxisRef) THEN
    RETURN;
END_IF

THIS^.AxisRef.ReadStatus();

(*Note: Configure within the axis parameters set "position correction" to true
    Directional change FOR compensation
      FALSE: positive backlash:
      TRUE -> Negative backlash compensation
    Reset Compensation to register a new value change
    fRampVelocity : a tenth of Moveabsolute velocity is a good starting point
*)
// use bUserBacklashEn for addtional control in user code, i.e fb_motionDrive
bLocalEnable R= NOT THIS^.bActive OR (THIS^.fBacklashComp<>THIS^.fPrevCompensation);
bLocalEnable S= THIS^.Error  AND THIS^.bActive;

fbMcBacklashCompensation(Axis:=AxisRef,
    Enable:= THIS^.bLocalEnable AND bUserEnable,
    Backlash:= THIS^.fBacklashComp,
    CompensationInPositiveDirection:=(THIS^.fBacklashComp < 0.0),
    Ramp:=( THIS^.fRampVelo ),
    DisableMode:=THIS^.eDisableMode,
    Enabled=> THIS^.bBacklashCompStatus,
    Error=>bError,
    ErrorID=>nErrorID,
    CurrentBacklash=>THIS^.fActCompensation
);
fPrevCompensation:=THIS^.fBacklashComp;

PROPERTY Aborted : BOOL
GET
END_GET
END_PROPERTY

{warning 'add property implementation'}
PROPERTY ActCompensation : LREAL
GET
ActCompensation := fActCompensation;
END_GET
END_PROPERTY

{warning 'Add property implementation'}
PROPERTY Active : BOOL
GET
END_GET
END_PROPERTY

(*
    Handle positive/negative backlash compensation
    User needs to set the direction of backlash from the sign of the compensation value
    Backlash compensation is disabled during referencing (homing).
    When direction is positive/negative, further movement in the negative/positive direction not compensated
    further movement in the negative/positive direction will be compensated
*)
METHOD BacklashCompensation
VAR_INPUT
    Activate     : BOOL;
    Compensation	: LREAL;
    RampVelocity	: LREAL;
    DisableMode	: E_DISABLEMODE := E_DISABLEMODE.DisableModeHold;
END_VAR
THIS^.bActive:= Activate;
THIS^.fBacklashComp := Compensation;
THIS^.fRampVelo := RampVelocity;
THIS^.eDisableMode:=DisableMode;
END_METHOD

(*synced Fbs need just to activate the compensation with a given ramp speed
  other parameters are provided via EPICS (declared in this FB) or via the more extended BackalshCompensation method (simulation) *)
METHOD BacklashCompensationActive
VAR_INPUT
    Active	: BOOL;
    RampVelocity	: LREAL;
END_VAR
THIS^.bActive:= Active;
THIS^.fRampVelo := RampVelocity;
END_METHOD

{warning 'Add property implementation'}
PROPERTY Busy : BOOL
GET
END_GET
END_PROPERTY

METHOD PUBLIC CallAfterInit
VAR_INPUT
    AxisRef : REFERENCE TO AXIS_REF;
END_VAR
THIS^.AxisRef REF= AxisRef;
END_METHOD

{warning 'Add property implementation'}
PROPERTY Done : BOOL
GET
END_GET
END_PROPERTY

PROPERTY Error : BOOL
GET
Error := bError;
END_GET
END_PROPERTY

PROPERTY ErrorID : UDINT
GET
ErrorID := nErrorID;
END_GET
END_PROPERTY

METHOD FB_Init : BOOL
VAR_INPUT
    bInitRetains : BOOL; // if TRUE, the retain variables are initialized (warm start / cold start)
    bInCopyCode : BOOL;  // if TRUE, the instance afterwards gets moved into the copy code (online change)
    AxisRef : REFERENCE TO AXIS_REF;
END_VAR
THIS^.AxisRef REF= AxisRef;
END_METHOD

PROPERTY Message : T_MaxString
GET
Message :=sMessage;
END_GET
END_PROPERTY

PROPERTY Status : BOOL
GET
Status := bBacklashCompStatus;
END_GET
END_PROPERTY

{warning 'Add property implementation'}
PROPERTY UserEnable : BOOL
SET
bUserEnable := UserEnable;
END_SET
END_PROPERTY

END_FUNCTION_BLOCK

// ---- POUs/FBs/NC/FB_ResetNC.TcPOU
FUNCTION_BLOCK FB_ResetNC IMPLEMENTS I_Reset
VAR
    {attribute 'no_copy'}
    AxisRef : REFERENCE TO AXIS_REF;
    fbMcReset 	: MC_Reset;
    bExecute : BOOL;
    bError : BOOL;
    bBusy : BOOL;
    bDone : BOOL;
    nErrorID : UDINT;
    sMessage : T_MAXSTRING;
    rtDone : R_TRIG;
    rtBusy : R_TRIG;
    btest : BOOL;
END_VAR

IF NOT __ISVALIDREF(THIS^.AxisRef) THEN
    RETURN;
END_IF

THIS^.AxisRef.ReadStatus();

THIS^.fbMcReset(
    Axis := THIS^.AxisRef,
    Execute := THIS^.bExecute (* AND Axis.Status.Error*),
    Done => THIS^.bDone,
    Busy => THIS^.bBusy,
    Error => THIS^.bError,
    ErrorID => THIS^.nErrorID,
);
rtBusy(CLK:=THIS^.bBusy);
IF rtBusy.Q THEN
    btest := TRUE;
END_IF
rtDone(CLK:=bDone);
IF  rtDone.Q THEN
    THIS^.bExecute := FALSE;
END_IF

{warning 'Add property implementation'}
PROPERTY Aborted : BOOL
GET
END_GET
END_PROPERTY

{warning 'Add property implementation'}
PROPERTY Active : BOOL
GET
END_GET
END_PROPERTY

PROPERTY Busy : BOOL
GET
Busy := bBusy;
END_GET
END_PROPERTY

